// enable elevation, enable azimuth
IF MAIN.ready AND CoverControl.isopen THEN
	ElevationControl.enable := TRUE;
	AzimuthElevationControl.enable := TRUE;
	DerotatorControl.enable := TRUE;
	FilterWheelControl.Enable := TRUE;
END_IF

IF ElevationControl.Ready AND NOT ElevationControl.Calibrated THEN
	ElevationControl.HomeAxis := TRUE;
END_IF

IF AzimuthElevationControl.ready AND NOT AzimuthElevationControl.calibrated THEN
	AzimuthElevationControl.HomeAxis := TRUE;
END_IF

// enable derotator
IF ElevationControl.Ready THEN
	DerotatorControl.HomeAxis := DerotatorControl.Ready AND NOT DerotatorControl.Calibrated;
END_IF

// home filterwheel after Derotator Axis to avoid additional torque
IF DerotatorControl.Calibrated THEN
	FilterWheelControl.HomeAxis := FilterWheelControl.Ready AND NOT FilterWheelControl.Calibrated;
END_IF

// start calibration of focus after elevation has been calibrated
// this avoids imbalance by the M2 mirror on the elvation during its calibration
IF ElevationControl.Calibrated AND NOT FocusControl.Calibrated THEN
	FocusControl.enable := TRUE;
	FocusControl.HomeAxis := TRUE;
END_IF

IF CoverControl.isopen AND 
	ElevationControl.Calibrated AND
	AzimuthElevationControl.calibrated AND
	DerotatorControl.Calibrated AND
	FilterWheelControl.Calibrated AND
	FocusControl.Calibrated THEN
	power := FALSE;
	poweron := TRUE;
	isparked := FALSE;
	// rest filterwheel until reactivation on filter change
	FilterWheelControl.Enable := FALSE;
	// slew the telescope to the home position
	gohome := TRUE;
ELSE
	poweron := FALSE;
END_IF
END_METHOD

METHOD slewtelescope : USINT
VAR_INPUT
END_VAR
VAR
	SlewEvent:	FB_Eventlog;
	command_timeout: TON;
END_VAR
VAR_STAT
	Stage:		USINT := 0;
	LastStage:	USINT := 101;
END_VAR
slewtelescope := Stage;
command_timeout(IN := Stage < 100, PT := T#600S);
IF command_timeout.Q THEN
	error := TRUE;
	errorid := 16#40;
	slew := FALSE;
	Stage := 0;
END_IF
IF reset OR error THEN
	Stage := 0;
END_IF
CASE Stage OF
	0:	
		IF ready AND stopped AND NOT busy AND NOT tracking THEN
			Stage := 25;
		END_IF
	25:
		ElevationControl.position := elevation;
		ElevationControl.velocity := 10.0;
		ElevationControl.MoveAxis := TRUE;
		AzimuthElevationControl.position := azimuth;
		AzimuthElevationControl.velocity := 10.0;
		AzimuthElevationControl.MoveAxis := TRUE;
		DerotatorControl.position := elevation + derotator_offset;
		DerotatorControl.Velocity := 10.0;
		DerotatorControl.MoveAxis := TRUE;
		IF ElevationControl.ElevationAxis.Busy AND
			AzimuthElevationControl.AzimuthAxis.Busy AND
			DerotatorControl.DerotatorAxis.Busy THEN
				Stage := 50;
		END_IF
	50:
		IF ElevationControl.ElevationAxis.MoveDone THEN
			ElevationControl.MoveAxis := FALSE;
		END_IF
		
		IF AzimuthElevationControl.AzimuthAxis.MoveDone THEN
			AzimuthElevationControl.MoveAxis := FALSE;
		END_IF

		IF DerotatorControl.DerotatorAxis.MoveDone THEN
			DerotatorControl.MoveAxis := FALSE;
		END_IF
		IF NOT sliding AND stopped THEN // all axis standstill
			Stage := 100;
		END_IF
	100:
		ElevationControl.MoveAxis := FALSE;
		AzimuthElevationControl.MoveAxis := FALSE;
		DerotatorControl.MoveAxis := FALSE;
		rightascension := rightascension_calc;
		declination := declination_calc;
		slew := FALSE;
		Stage := 0;
END_CASE
SlewEvent(Trigger := Stage > LastStage, FormatString := 'Slew progress: %s', OnMessage := USINT_TO_STRING(Stage));
LastStage := Stage;
END_METHOD

METHOD stoptelescope : BOOL
VAR_INPUT
END_VAR
ElevationControl.StopAxis := TRUE;
AzimuthElevationControl.StopAxis := TRUE;
DerotatorControl.StopAxis := TRUE;
IF stopped THEN
	ElevationControl.StopAxis := FALSE;
	AzimuthElevationControl.StopAxis := FALSE;
	DerotatorControl.StopAxis := FALSE;
	stop := FALSE;
END_IF
END_METHOD

METHOD tracktelescope : BOOL
VAR_INPUT
END_VAR
// Elevation
DerotatorVelocity := F_Derotatorvelocity(elevation_calc, azimuth_calc, latitude);
ElevationVelocity := F_Elevationvelocity(azimuth_calc, latitude);
AzimuthVelocity := F_Azimuthvelocity(elevation_calc, azimuth_calc, latitude);
IF elevation_current < 5.0 OR elevation_current > 89.5 THEN 
	track := FALSE;
END_IF
IF azimuth_current > 440.0 THEN
	track := FALSE;
END_IF
IF (derotator_current < -69.0 AND DerotatorVelocity<0.0) OR (derotator_current > 379.0 AND DerotatorVelocity>0.0) THEN
	track := FALSE;
END_IF

ElevationControl.position := elevation_calc;
IF NOT ElevationControl.Tracking THEN
	ElevationControl.velocity := 10.0;
	ElevationControl.MoveAxis := TRUE;
	IF NOT ElevationControl.ElevationAxis.Busy AND ElevationControl.ElevationAxis.MoveDone THEN
		ElevationControl.MoveAxis := FALSE;
		IF ElevationControl.ElevationAxis.isTracking THEN
			ElevationControl.velocity := ElevationVelocity;
		ELSE
			ElevationControl.velocity := 3.0*ElevationVelocity;
		END_IF
		ElevationControl.velocity := ElevationVelocity;
		ElevationControl.Tracking := TRUE;
	END_IF
ELSE
	ElevationControl.velocity := ElevationVelocity;
END_IF

// Azimuth
AzimuthElevationControl.position := azimuth_calc;
IF NOT AzimuthElevationControl.Tracking THEN
	AzimuthElevationControl.velocity := 10.0;
	AzimuthElevationControl.MoveAxis := TRUE;
	IF NOT AzimuthElevationControl.AzimuthAxis.Busy AND AzimuthElevationControl.AzimuthAxis.MoveDone THEN
		AzimuthElevationControl.MoveAxis := FALSE;
		IF AzimuthElevationControl.AzimuthAxis.isTracking THEN
			AzimuthElevationControl.velocity := AzimuthVelocity;
		ELSE
			AzimuthElevationControl.velocity := 3.0*AzimuthVelocity;
		END_IF
		AzimuthElevationControl.velocity := AzimuthVelocity;
		AzimuthElevationControl.Tracking := TRUE;
	END_IF
ELSE
	AzimuthElevationControl.velocity := AzimuthVelocity;
END_IF

// Derotator
DerotatorControl.position := derotation_calc;
IF NOT DerotatorControl.Tracking THEN
	DerotatorControl.Velocity := 10.0;
	DerotatorControl.MoveAxis := TRUE;
	IF NOT DerotatorControl.DerotatorAxis.Busy AND DerotatorControl.DerotatorAxis.MoveDone THEN
		DerotatorControl.MoveAxis := FALSE;
		IF DerotatorControl.DerotatorAxis.isTracking THEN
			DerotatorControl.Velocity := DerotatorVelocity;
		ELSE
			DerotatorControl.Velocity := 3.0*DerotatorVelocity;
		END_IF
		DerotatorControl.Velocity := DerotatorVelocity;
		DerotatorControl.Tracking := TRUE;
	END_IF
ELSE
	DerotatorControl.Velocity := DerotatorVelocity;
END_IF
END_METHOD

END_PROGRAM

// ---- POUs/FunctionBlocks/FB_AstroClock.TcPOU
FUNCTION_BLOCK FB_AstroClock
VAR_INPUT
END_VAR
VAR_OUTPUT
        time_RTCEX      : DT;
        time_RTCEX2     : TIMESTRUCT;
        nMilliseconds   : DWORD;
        nMicroseconds   : DWORD;
END_VAR
VAR
	        fbGetLocalTime  : NT_GetTime;
        bBusy           : BOOL;
        bError          : BOOL;
        nErrID          : UDINT;
        presetTime      : TIMESTRUCT;

        syncTimer       : TON;
        syncTrigger     : F_TRIG;
        bSynchronize    : BOOL;

        fbRTC           : RTC;
        bValid_RTC      : BOOL;
        time_RTC        : DT;

        fbRTC_EX        : RTC_EX;
        bValid_RTCEX    : BOOL;

        fbRTC_EX2       : RTC_EX2;
        bValid_RTCEX2   : BOOL;
END_VAR

(*
TYPE TIMESTRUCT
STRUCT
   wYear            : WORD;
   wMonth           : WORD;
   wDayOfWeek       : WORD;
   wDay             : WORD;
   wHour            : WORD;
   wMinute          : WORD;
   wSecond          : WORD;
   wMilliseconds    : WORD;
END_STRUCT
END_TYPE
*)

syncTimer(IN := NOT SyncTimer.Q, PT := T#5S);
fbGetLocalTime(START := syncTimer.Q,
	TMOUT := DEFAULT_ADS_TIMEOUT,
	Busy => bBusy,
	ERR => bError,
	ERRID => nErrID,
	TIMESTR => presetTime);

syncTrigger(CLK := bBusy AND NOT bError, Q => bSynchronize);

fbRTC(EN := bSynchronize,
	PDT := SYSTEMTIME_TO_DT(presetTime),
	Q => bValid_RTC,
	CDT => time_RTC);
	
fbRTC_EX(EN := bSynchronize,
	PDT := SYSTEMTIME_TO_DT(presetTime),
	PMSEK := presetTime.wMilliseconds,
	Q => bValid_RTCEX,
	CDT => time_RTCEX,
	CMSEK => nMilliseconds);

fbRTC_EX2(EN := bSynchronize,
	PDT := presetTime,
	PMICRO := 0,
	Q => bValid_RTCEX2,
	CDT => time_RTCEX2,
	CMICRO => nMicroseconds);

END_FUNCTION_BLOCK

// ---- POUs/FunctionBlocks/FB_EQ2HOR2.TcPOU
FUNCTION_BLOCK FB_EQ2HOR2
VAR_INPUT
	// right ascension in degrees
	alpha: LREAL;
	// declination in degrees
	delta: LREAL;
	// longitude in degrees
	lon: LREAL;
	// latitude in degrees
	lat: LREAL;
	// Julian Days
	JD: LREAL;
END_VAR
VAR_OUTPUT
	// altitude in degrees
	alt: LREAL;
	// azimuth in degrees
	az: LREAL;
	// hour angle in degreesss
	ha: LREAL;
END_VAR
VAR
	lst: LREAL;
	// helper variables
	sinalt,
	// in radians
	phi_r, tau_r, alpha_r, delta_r: LREAL;
	// current epoch
	J_now: 		LREAL;
	// enable precession
	precess: 	BOOL := TRUE;
	// enable nutation
	nutate:		BOOL := TRUE;
	// enable abberation
	abberation:	BOOL := TRUE;
	// enable refraction correction
	refract:	BOOL := TRUE;
	// precession function block
	fbprecess: 	FB_PRECESS3;
	// nutation function block
	co_nutate: CO_NUTATE;
	// abberration function block
	fbaberration: CO_ABERRATION;
	//precessed coordinates
	alpha1, delta1, 
	d_alpha2, d_delta2, 
	d_alpha3, d_delta3:	LREAL;
END_VAR
VAR CONSTANT
	d2r:	LREAL := PI/180.0;
	r2d:	LREAL := 180.0/PI;
END_VAR

(* 
source: http://star-www.st-and.ac.uk/~fv/webnotes/chapter7.htm
https://squarewidget.com/astronomical-calculations-sidereal-time/

*)
lst := ct2lst(lon, jd) * 15.0; // lst in degrees

J_now := (JD - 2451545.0)/365.25 + 2000.0; // compute current equinox
IF precess THEN
	fbprecess( ra := alpha, dec := delta, 
	//EQUINOX1 := 2000.0, EQUINOX2 := J_now, 
	ra_precessed =>alpha1, dec_precessed => delta1);
ELSE
	alpha1 := alpha;
	delta1 := delta;	
END_IF

IF nutate THEN
	co_nutate(	jd := jd, 
				ra := alpha, 
				dec := delta, 
				d_ra => d_alpha2, 
				d_dec => d_delta2);
	alpha1 := alpha1 + d_alpha2;
	delta1 := delta1 + d_delta2;
ELSE
	d_alpha2 := 0.0;
	d_delta2 := 0.0;
END_IF

IF abberation THEN
	fbaberration(	jd := jd, 
					ra := alpha, 
					dec := delta, 
					d_ra => d_alpha3, 
					d_dec => d_delta3);
	alpha1 := alpha1 + d_alpha3;
	delta1 := delta1 + d_delta3;
ELSE
	d_alpha3 := 0.0;
	d_delta3 := 0.0;
END_IF

ha := MODABS(lst - alpha1, 360.0);

alpha_r := alpha1 * d2r;
delta_r := delta1 * d2r;
tau_r := lst*d2r - alpha_r;
phi_r := lat*d2r;

sinalt := SIN(phi_r)*SIN(delta_r) + COS(phi_r)*COS(delta_r)*COS(tau_r);
alt := ASIN(sinalt) * r2d;
IF refract THEN
	alt := alt + Refraction(alt, pressure := 770.0, temperature := 10.0);
END_IF
az := ATAN2(SIN(tau_r), SIN(phi_r)*COS(tau_r) - COS(phi_r)*TAN(delta_r)) * r2d + 180.0;

END_FUNCTION_BLOCK

// ---- POUs/FunctionBlocks/FB_PRECESS3.TcPOU
FUNCTION_BLOCK FB_PRECESS3
VAR_INPUT
	// right ascension in degrees
	ra: LREAL;
	// declination in degrees
	dec: LREAL;
	
END_VAR
VAR_OUTPUT
	// precessed right ascension
	ra_precessed:	LREAL;
	// precessed declination
	dec_precessed:	LREAL;
END_VAR
VAR
	ra_rad, dec_rad: LREAL;
	// starting jd (J2000)
	jd0: LREAL;
	// traget JD
	jd: LREAL;
	t, 
	eta, 
	z, 
	phi,
	A,
	B,
	C	: LREAL;
END_VAR
VAR CONSTANT
	deg_to_rad : LREAL := PI/180.0;
	sec_to_rad : LREAL := deg_to_rad/3600.0;
END_VAR

// see Jean Meeus p.135

ra_rad := ra*deg_to_rad;
dec_rad := dec*deg_to_rad;

// todo epoch to jd and jd0
JD := TelescopeControl.jd;
jd0 := 2451545.0;
t := (jd - jd0) / 36525.0;

eta :=	(2306.2181*t + 0.30188*t*t + 0.017998*t*t*t) * sec_to_rad;
z :=	(2306.2181*t + 1.09468*t*t + 0.018203*t*t*t) * sec_to_rad;
phi :=	(2004.3109*t - 0.42665*t*t - 0.041833*t*t*t) * sec_to_rad;

A :=            COS(dec_rad) * SIN(ra_rad + eta);
B := COS(phi) * COS(dec_rad) * COS(ra_rad + eta) - SIN(phi) * SIN(dec_rad);
C := SIN(phi) * COS(dec_rad) * COS(ra_rad + eta) + COS(phi) * SIN(dec_rad);

// tan(ra - z) == A/B
ra_precessed := MODABS((ATAN2(A, B) + z)/deg_to_rad, 360);
IF ABS(dec) > 89.5 THEN
	dec_precessed := ACOS(SQRT(A*A + B*B))/deg_to_rad;
ELSE
	// sin(de)c = C
	dec_precessed := ASIN(C)/deg_to_rad;	
END_IF

END_FUNCTION_BLOCK

// ---- POUs/Functions/ATAN2.TcPOU
FUNCTION ATAN2 : LREAL
VAR_INPUT
	y, x: LREAL;
END_VAR
VAR
END_VAR

(* source: https://de.wikipedia.org/wiki/Arctan2 
arctan2(y, x) := arctan(x/y)*sgn(x)^2
WARNING! The arguments are reversed compared to original wiki formula!
 *)
ATAN2 := 0.0;

IF x > 0 THEN
	ATAN2 := ATAN(y/x);
ELSIF x < 0 AND y > 0 THEN
	ATAN2 := ATAN(y/x) + PI;
ELSIF x < 0 AND y = 0 THEN
	ATAN2 := PI;
ELSIF x < 0 AND y < 0 THEN
	ATAN2 := ATAN(y/x) - PI;
ELSIF x = 0 AND y > 0 THEN
	ATAN2 := PI/2.0;
ELSIF x = 0 AND y < 0 THEN
	ATAN2 := -PI/2.0;
END_IF

END_FUNCTION

// ---- POUs/FunctionBlocks/CO_NUTATE.TcPOU
FUNCTION_BLOCK CO_NUTATE
VAR_INPUT
	// Julian date
	jd:	LREAL;
	// right ascension
	ra: LREAL;
	// declination
	dec: LREAL;
END_VAR
VAR_OUTPUT
	d_ra:	LREAL;
	d_dec:	LREAL;
	eps:	LREAL;
	d_psi:	LREAL;
END_VAR
VAR
	T, eps0, d_eps, ce, se, x,y,z, ra2, dec2: LREAL;
	x2, y2, z2:	LREAL;
	radius, xyproj: 	LREAL;
	nutate:	FB_NUTATE;
END_VAR
VAR CONSTANT
	d2r:	LREAL := PI/180.0;
	d2as: 	LREAL := PI/(180.0*3600.0);
END_VAR

 
T := (jd - 2451545.0)/36525.0; // Julian centuries FROM J2000 OF jd.

// must calculate obliquity of ecliptic
nutate(jd := jd, nut_long => d_psi, nut_obliq => d_eps );

eps0 := 23.4392911*3600.0 - 46.8150*T - 0.00059*T*T + 0.001813*T*T*T;
eps := (eps0 + d_eps)/3600.0*d2r; // true obliquity of the ecliptic in radians
 
//useful numbers
ce := COS(eps);
se := SIN(eps);

// convert ra-dec to equatorial rectangular coordinates
x := COS(ra*d2r) * COS(dec*d2r);
y := SIN(ra*d2r) * COS(dec*d2r);
z := SIN(dec*d2r);

// apply corrections to each rectangular coordinate
x2 := x - (y*ce + z*se)*d_psi * d2as;
y2 := y + (x*ce*d_psi - z*d_eps) * d2as;
z2 := z + (x*se*d_psi + y*d_eps) * d2as;

// convert back to equatorial spherical coordinates
radius := SQRT(x2*x2 + y2*y2 + z2*z2);
xyproj := SQRT(x2*x2 + y2*y2);

ra2 := x2 * 0.0;
dec2:= x2 * 0.0;
// Calculate Ra and Dec in RADIANS (later convert to DEGREES)

IF xyproj = 0.0 AND z <> 0.0 THEN
	// places where xyproj:=0 (point at NCP or SCP)
	dec2 := ASIN(z2/radius);
	ra2 := 0.0;
END_IF
IF xyproj <> 0.0 THEN
	ra2 := ATAN2(y2, x2);
	dec2 := ASIN(z2 / radius);
END_IF

// convert to DEGREES
ra2 := ra2 /d2r;
dec2 := dec2 /d2r;

// w := where(ra2 LT 0., Nw)
// IF Nw GT 0 THEN ra2[w] := ra2[w] + 360.
ra2 := MODABS(ra2, 360.0);

// Return changes in ra and dec in degrees
 d_ra := ra2 - ra;
 d_dec := dec2 - dec;

END_FUNCTION_BLOCK

// ---- POUs/FunctionBlocks/FB_NUTATE.TcPOU
FUNCTION_BLOCK FB_NUTATE
VAR_INPUT
	jd:	LREAL;
END_VAR
VAR_OUTPUT
	nut_long, nut_obliq: LREAL := 0.0;
END_VAR
VAR
	t: LREAL;
	d, M, Mprime, F, omega: LREAL;
	arg, sarg, carg:  ARRAY[0..62] OF LREAL;
	I: INT;
END_VAR
VAR CONSTANT
	dtor:	LREAL := PI/180.0;
	coeff1:	ARRAY[0..3] OF LREAL := [297.85036, 445267.111480, -0.0019142,  1.0/189474];
	coeff2:	ARRAY[0..3] OF LREAL := [357.52772,  35999.050340, -0.0001603, -1.0/3E5]; 
	coeff3:	ARRAY[0..3] OF LREAL := [134.96298, 477198.867398,  0.0086972,  1.0/5.625E4]; 
	coeff4:	ARRAY[0..3] OF LREAL :=  [93.27191, 483202.017538, -0.0036825, -1.0/3.27270E5]; 
  	coeff5: ARRAY[0..3] OF LREAL := [125.04452,  -1934.136261,  0.0020708,  1.0/4.5E5];
	d_lng: ARRAY[0..62] OF LREAL := [0,-2,0,0,0,0,-2,0,0,-2,-2,-2,0,2,0,2,0,0,-2,0,2,0,0,-2,0,-2,0,0,2,-2,0,-2,0,0,2,2,0,-2,0,2,2,-2,-2,2,2,0,-2,-2,0,-2,-2,0,-1,-2,1,0,0,-1,0,0,2,0,2]; 
	m_lng: ARRAY[0..62] OF LREAL := [0,0,0,0,1,0,1,0,0,-1,17(0),2,0,2,1,0,-1,0,0,0,1,1,-1,0,0,0,0,0,0,-1,-1,0,0,0,1,0,0,1,0,0,0,-1,1,-1,-1,0,-1];
	mp_lng: ARRAY[0..62] OF LREAL := [0,0,0,0,0,1,0,0,1,0,1,0,-1,0,1,-1,-1,1,2,-2,0,2,2,1,0,0,-1,0,-1,0,0,1,0,2,-1,1,0,1,0,0,1,2,1,-2,0,1,0,0,2,2,0,1,1,0,0,1,-2,1,1,1,-1,3,0];
	f_lng: ARRAY[0..62] OF LREAL := [0,2,2,0,0,0,2,2,2,2,0,2,2,0,0,2,0,2,0,2,2,2,0,2,2,2,2,0,0,2,0,0,0,-2,2,2,2,0,2,2,0,2,2,0,0,0,2,0,2,0,2,-2,0,0,0,2,2,0,0,2,2,2,2];
	om_lng: ARRAY[0..62] OF LREAL := [1,2,2,2,0,0,2,1,2,2,0,1,2,0,1,2,1,1,0,1,2,2,0,2,0,0,1,0,1,2,1,1,1,0,1,2,2,0,2,1,0,2,1,1,1,0,1,1,1,1,1,0,0,0,0,0,2,0,0,2,2,2,2];
	sin_lng: ARRAY[0..62] OF LREAL := [-171996, -13187, -2274, 2062, 1426, 712, -517, -386, -301, 217, -158, 129, 123, 63, 63, -59, -58, -51, 48, 46, -38, -31, 29, 29, 26, -22, 21, 17, 16, -16, -15, -13, -12, 11, -10, -8, 7, -7, -7, -7, 6,6,6,-6,-6,5,-5,-5,-5,4,4,4,-4,-4,-4,3,-3,-3,-3,-3,-3,-3,-3 ];
	sdelt: ARRAY[0..62] OF LREAL := [-174.2, -1.6, -0.2, 0.2, -3.4, 0.1, 1.2, -0.4, 0, -0.5, 0, 0.1, 0,0,0.1, 0,-0.1,10(0), -0.1, 0, 0.1, 33(0)];
	cos_lng: ARRAY[0..62] OF LREAL := [ 92025, 5736, 977, -895, 54, -7, 224, 200, 129, -95,0,-70,-53,0, -33, 26, 32, 27, 0, -24, 16,13,0,-12,0,0,-10,0,-8,7,9,7,6,0,5,3,-3,0,3,3, 0,-3,-3,3,3,0,3,3,3, 14(0)] ;
	cdelt: ARRAY[0..62] OF LREAL := [8.9, -3.1, -0.5, 0.5, -0.1, 0.0, -0.6, 0.0, -0.1, 0.3, 53(0)];
END_VAR

//  form time in Julian centuries from 1900.0

t := (jd - 2451545.0)/36525.0;

// Mean elongation of the Moon

d := poly(T, coeff1)*dtor;
d := MODABS(d, 2.0*PI);

// Sun's mean anomaly

M := poly(T,coeff2)*dtor;
M := MODABS(M, 2.0*PI);

// Moon's mean anomaly

Mprime := poly(T,coeff3)*dtor;
Mprime := MODABS(Mprime, 2.0*PI);

// Moon's argument of latitude

F := poly(T, coeff4 )*dtor;
F := MODABS(F, 2.0*PI);

// Longitude OF the ascending node OF the Moon's mean orbit on the ecliptic,
//  measured from the mean equinox of the date

omega := poly(T, coeff5)*dtor;
omega := MODABS(omega, 2.0*PI);


// Sum the periodic terms 
FOR i:=0 TO 62 DO
	arg[i] := d_lng[i]*d + m_lng[i]*m +mp_lng[i]*mprime + f_lng[i]*f +om_lng[i]*omega;
	sarg[i] := SIN(arg[i]);
	carg[i] := COS(arg[i]);
END_FOR

nut_long  := 0.0;
nut_obliq := 0.0;

FOR i:=0 TO 62 DO
	nut_long  := nut_long  + 0.0001*( (sdelt[i]*t + sin_lng[i])*sarg[i]);
	nut_obliq := nut_obliq + 0.0001*( (cdelt[i]*t + cos_lng[i])*carg[i]);
END_FOR

END_FUNCTION_BLOCK

// ---- POUs/Functions/POLY.TcPOU
FUNCTION POLY : LREAL
VAR_INPUT
	X:	LREAL;
	COEFFS: ARRAY [0..3] OF LREAL;
END_VAR
VAR
END_VAR

POLY := COEFFS[0]*EXPT(X, 0) + COEFFS[1]*EXPT(X, 1) + COEFFS[2]*EXPT(X, 2) + COEFFS[3]*EXPT(X, 3);

END_FUNCTION

// ---- POUs/FunctionBlocks/CO_ABERRATION.TcPOU
FUNCTION_BLOCK CO_ABERRATION
VAR_INPUT
	jd, 				// Julian Date
	ra, dec: LREAL; 	//ra and dec in degrees
	eps : LREAL := 0.0;
END_VAR
VAR_OUTPUT
	d_ra, d_dec: LREAL;
END_VAR
VAR
	sunpos: FB_SUNPOS;
	nutate: FB_NUTATE;
	sunra, sundec, sunlon,
	d_psi, d_epsilon, eps0,
	t, e, peri, cd, sd, ce, te, cp, sp, cs, ss, ca, sa, term1, term2, term3, term4: LREAL;
END_VAR
VAR CONSTANT
	d2r : LREAL := PI/180.0;
	k: LREAL := 20.49552; //constant of aberration, in arcseconds
	
END_VAR

(*
;+
;  NAME:
;     CO_ABERRATION
; PURPOSE:
;     Calculate changes to Ra and Dec due to the effect of annual aberration 
; EXPLANATION:
;      as described in Meeus, Chap 23.
; CALLING SEQUENCE:
;      co_aberration, jd, ra, dec, d_ra, d_dec, [EPS = ]
; INPUTS
;       jd      : Julian Date [scalar or vector]
;       ra, dec : Arrays (or scalars) of the ra  and dec's in degrees
;   Note: if jd is a vector, then ra and dec must either be scalars, or 
;                vectors of the same length.
;
; OUTPUTS
;       d_ra, d_dec: the corrections to ra and dec due to aberration in 
;                    arcseconds.  (These values can be added to the true RA 
;                    and dec to get the apparent position).   Note that d_ra
;                     is *not* multiplied by cos(dec), so that 
;                     apparent_ra = ra + d_ra/3600. 
; OPTIONAL INPUT KEYWORD:
;       eps : set this to the true obliquity of the ecliptic (in radians), or
;         it will be set for you if you don't know it (in that case, set it to
;                 an empty variable).
; EXAMPLE:
;   Compute the change in RA and Dec of Theta Persei (RA = 2h46m,11.331s, Dec =
;   49d20',54.54") due to aberration on 2028 Nov 13.19 TD
;
;      IDL> jdcnv,2028,11,13,.19*24,jd      ;Get Julian date
;      IDL> co_aberration,jd,ten(2,46,11.331)*15,ten(49,20,54.54),d_ra,d_dec
;
;      ==> d_ra = 30.045" (=2.003s)    d_dec = 6.697"
; NOTES:
;  These formula are from Meeus, Chapters 23.  Accuracy is much better than 1 
;   arcsecond.
;
;   The maximum deviation due to annual aberration is 20.49" and occurs when the
;   Earth velocity is perpendicular to the direction of the star.
;
; REVISION HISTORY:
;   Written, June 2002,      Chris O'Dell, U. of Wisconsin
;   Fix error with vector input   W. Landsman   June 2009
;   June 2009 update fixed case where JD was scalar but RA,Dec were vectors, but 
;     broke the case when both JD and RA,Dec were vectors Aug 2012 W. Landsman
;   Further fix when JD is 1 element vector  W. Landsman
;-
*)

T := (jd -2451545.0)/36525.0; // julian centuries from J2000 of jd.

IF EPS = 0.0 THEN
	// must calculate obliquity of ecliptic
	nutate(jd := jd, nut_long => d_psi, nut_obliq => d_epsilon); //d_psi and d_epsilon in degrees
	eps0 := ten(23,26,21.448)*3600.0 - 46.8150*T - 0.00059*EXPT(T, 2) +  0.001813*EXPT(T, 3);
	// TRUE obliquity OF the ecliptic in radians
	eps := (eps0 + d_epsilon)/3600.0*d2r; 	
END_IF

sunpos( JD := jd, RA => sunra, Dec => sundec, longmed => sunlon);

// Earth's orbital eccentricity
e := 0.016708634 - 0.000042037*T - 0.0000001267*EXPT(T, 2);
// longitude of perihelion, in degrees 
peri := 102.93735 + 1.71946*T + 0.00046*EXPT(T, 2);

//Useful Trig Functions
cd := COS(dec*d2r);		sd := SIN(dec*d2r);
ce := COS(eps); 		te := TAN(eps);
cp := COS(peri*d2r);	sp := SIN(peri*d2r);
cs := COS(sunlon*d2r);	ss := SIN(sunlon*d2r);
ca := COS(ra*d2r);		sa := SIN(ra*d2r);

term1 := (ca*cs*ce + sa*ss)/cd;
term2 := (ca*cp*ce + sa*sp)/cd;
term3 := (cs*ce*(te*cd - sa*sd) + ca*sd*ss);
term4 := (cp*ce*(te*cd - sa*sd) + ca*sd*sp);

d_ra := (-k * term1 + e*k * term2)/3600.0;
d_dec := (-k * term3 + e*k * term4)/3600.0;

END_FUNCTION_BLOCK

// ---- POUs/FunctionBlocks/FB_SUNPOS.TcPOU
FUNCTION_BLOCK FB_SUNPOS
VAR_INPUT
	// Julian Date
	JD:		LREAL;
	// output in Radians instead of Degrees
	RADIAN:	BOOL:= FALSE;
END_VAR
VAR_OUTPUT
	// right ascension
	RA,
	// declination of the sun
	Dec,
	// longitude
	longmed,
	// True Obliquity
	oblt:	LREAL;
END_VAR
VAR
	t, //  Julian centuries FROM 1900.0
	l, //  sun's mean longitude
	me, // Earth's mean anomaly
	ellcor, // ellipticity of the orbit
	mv, // mean anomaly of Venus
	vencorr,
	mm, 
	marscorr,
mj, jupcorr,
d, longterm, mooncorr,  omega:	LREAL;
END_VAR
VAR CONSTANT
	dtor: LREAL := PI/180.0; // Pi/180
END_VAR

(* source: https://idlastro.gsfc.nasa.gov/ftp/pro/astro/sunpos.pro *)

//  form TIME in Julian centuries FROM 1900.0
t := (jd - 2415020.0)/36525.0;

//  form sun's mean longitude
l := (279.696678+LMOD(36000.768925*t, 360.0))*3600.0;

//  allow for ellipticity of the orbit (equation of centre) using the Earth's mean anomaly ME
me := 358.475844 + LMOD(35999.049750*t, 360.0);
ellcor  := (6910.1 - 17.2*t)*SIN(me*dtor) + 72.3*SIN(2.0*me*dtor);
l := l + ellcor;
 
// allow FOR the Venus perturbations using the mean anomaly OF Venus MV
mv := 212.603219 + LMOD(58517.803875*t, 360.0);
vencorr := 4.8 * COS((299.1017 + mv - me)*dtor) + 
          5.5 * COS((148.3133 +  2.0 * mv  -  2.0 * me )*dtor) + 
          2.5 * COS((315.9433 +  2.0 * mv  -  3.0 * me )*dtor) + 
          1.6 * COS((345.2533 +  3.0 * mv  -  4.0 * me )*dtor) + 
          1.0 * COS((318.15   +  3.0 * mv  -  5.0 * me )*dtor);
l := l + vencorr;

//  Allow FOR the Mars perturbations using the mean anomaly OF Mars MM
mm := 319.529425  +  LMOD( 19139.858500 * t,  360.0 );
marscorr := 2.0 * COS((343.8883 -  2.0 * mm  +  2.0 * me)*dtor ) + 
            1.8 * COS((200.4017 -  2.0 * mm  + me) * dtor);
l := l + marscorr;

// Allow FOR the Jupiter perturbations using the mean anomaly OF Jupiter MJ
mj := 225.328328  +  LMOD( 3034.6920239 * t,  360.0 );
jupcorr := 7.2 * COS(( 179.5317 - mj + me )*dtor) + 
          2.6 * COS((263.2167  -  MJ ) *dtor) + 
          2.7 * COS(( 87.1450  -  2.0 * mj  +  2.0 * me ) *dtor) + 
          1.6 * COS((109.4933  -  2.0 * mj  +  me ) *dtor);
l := l + jupcorr;

// Allow FOR the Moons perturbations using the mean elongation OF the Moon from the Sun D
d := 350.7376814  + LMOD( 445267.11422 * t,  360.0 );
mooncorr  := 6.5 * SIN(d*dtor);
l := l + mooncorr;

// Allow for long period terms
longterm := 6.4 * SIN(( 231.19  +  20.20 * t )*dtor);
l :=  l + longterm;
l :=  LMOD( l + 2592000.0,  1296000.0); 
longmed := l/3600.0;

// Allow for Aberration
l :=  l - 20.5;

// Allow for Nutation using the longitude of the Moons mean node OMEGA
omega := 259.183275 - LMOD( 1934.142008 * t, 360.0);
l :=  l - 17.2 * SIN(omega*dtor);

// Form the True Obliquity
oblt := 23.452294 - 0.0130125*t + (9.2*COS(omega*dtor))/3600.0;

// Form Right Ascension AND Declination
l := l/3600.0;
ra := ATAN2( SIN(l*dtor) * COS(oblt*dtor), COS(l*dtor));
//ra := MODABS(ra, 360.0);
dec := ASIN(SIN(l*dtor) * SIN(oblt*dtor));
 
IF RADIAN THEN
	oblt := oblt*dtor; 
	longmed := longmed*dtor;
ELSE
	ra := ra/dtor;
    dec := dec/dtor;
END_IF

END_FUNCTION_BLOCK

// ---- POUs/Functions/CT2LST.TcPOU
FUNCTION CT2LST : LREAL
VAR_INPUT
	lng: LREAL; // The longitude in degrees (east of Greenwich) of the place for which the local sidereal time is desired, scalar.   The Greenwich mean sidereal time (GMST) can be found by setting Lng = 0.
	jd:	LREAL; // this is the Julian date of time in question
END_VAR
VAR
	t0,t,theta: LREAL;
END_VAR
VAR CONSTANT
	jd2000: LREAL := 2451545.0;
END_VAR

(* source https://idlastro.gsfc.nasa.gov/ftp/pro/astro/ct2lst.pro 

;+
; NAME:
;     CT2LST
; PURPOSE:
;     To convert from Local Civil Time to Local Mean Sidereal Time.
;
; CALLING SEQUENCE:
;     CT2LST, Lst, Lng, Tz, Time, [Day, Mon, Year] 
;                       or
;     CT2LST, Lst, Lng, dummy, JD
;
; INPUTS:
;     Lng  - The longitude in degrees (east of Greenwich) of the place for 
;            which the local sidereal time is desired, scalar.   The Greenwich 
;            mean sidereal time (GMST) can be found by setting Lng = 0.
;     Tz  - The time zone of the site in hours, positive East  of the Greenwich
;           meridian (ahead of GMT).  Use this parameter to easily account 
;           for Daylight Savings time (e.g. -4=EDT, -5 = EST/CDT), scalar
;           This parameter is not needed (and ignored) if Julian date is 
;           supplied.    ***Note that the sign of TZ was changed in July 2008
;           to match the standard definition.*** 
;     Time or JD  - If more than four parameters are specified, then this is 
;               the time of day of the specified date in decimal hours.  If 
;               exactly four parameters are specified, then this is the 
;               Julian date of time in question, scalar or vector
;
; OPTIONAL INPUTS:
;      Day -  The day of the month (1-31),integer scalar or vector
;      Mon -  The month, in numerical format (1-12), integer scalar or vector
;      Year - The 4 digit year (e.g. 2008), integer scalar or vector
;
; OUTPUTS:
;       Lst   The Local Sidereal Time for the date/time specified in hours.
;
; RESTRICTIONS:
;       If specified, the date should be in numerical form.  The year should
;       appear as yyyy.
;
; PROCEDURE:
;       The Julian date of the day and time is question is used to determine
;       the number of days to have passed since 0 Jan 2000.  This is used
;       in conjunction with the GST of that date to extrapolate to the current
;       GST; this is then used to get the LST.    See Astronomical Algorithms
;       by Jean Meeus, p. 84 (Eq. 11-4) for the constants used.
;
; EXAMPLE:
;       Find the Greenwich mean sidereal time (GMST) on 2008 Jul 30 at 15:53 pm
;       in Baltimore, Maryland (longitude=-76.72 degrees).   The timezone is 
;       EDT or tz=-4
;
;       IDL> CT2LST, lst, -76.72, -4,ten(15,53), 30, 07, 2008
;
;               ==> lst =  11.356505  hours  (= 11h 21m 23.418s)
;
;       The Web site  http://tycho.usno.navy.mil/sidereal.html contains more
;       info on sidereal time, as well as an interactive calculator.
; PROCEDURES USED:
;       jdcnv - Convert from year, month, day, hour to julian date
;
; MODIFICATION HISTORY:
;     Adapted from the FORTRAN program GETSD by Michael R. Greason, STX, 
;               27 October 1988.
;     Use IAU 1984 constants Wayne Landsman, HSTX, April 1995, results 
;               differ by about 0.1 seconds  
;     Longitudes measured *east* of Greenwich   W. Landsman    December 1998
;     Time zone now measure positive East of Greenwich W. Landsman July 2008
;     Remove debugging print statement  W. Landsman April 2009
;-

*)

t0 := jd - jd2000;
t := t0/36525.0;
// Compute GST in seconds.
theta := 280.46061837 + (360.98564736629 * t0) + EXPT(t, 2)*(0.000387933 - (t/ 3871.0E4));
//theta := 100.46061837 + 36000.770053608*t0 + 0.000387933*EXPT(t0,2) - EXPT(t0,3)/3871000.0;
// Compute LST in hours.
CT2LST := ( theta + lng)/15.0;
CT2LST := MODABS(CT2LST, 24.0);

END_FUNCTION

// ---- POUs/Functions/Refraction.TcPOU
FUNCTION Refraction : LREAL
VAR_INPUT
	// elevation in degrees
	elevation: LREAL;
	// pressure in mBar
	pressure: LREAL := 770.0;
	// temperature in Celsius
	temperature : LREAL := 10.0;
END_VAR
VAR
END_VAR
VAR CONSTANT
	d2r:	LREAL := PI/180.0;
END_VAR

// sanity checks
elevation := LIMIT(0.0, elevation, 90.0);
pressure := LIMIT(600.0, pressure, 1200.0);
temperature := LIMIT(-30.0, temperature, 40.0);
// refraction in arcmin
Refraction := 1.02 / TAN((elevation + 10.3/(elevation + 5.11)) * d2r);
Refraction := Refraction * pressure * 283.0 / (1010.0 * (273.0 + temperature));
//refraction in degrees
Refraction := Refraction / 60.0;

END_FUNCTION

// ---- POUs/FunctionBlocks/FB_HOR2EQ.TcPOU
FUNCTION_BLOCK FB_HOR2EQ
VAR_INPUT
	//altitude (in degrees) [scalar OR vector]
	alt: LREAL;  
	//azimuth angle (in degrees, measured EAST from NORTH, but see keyword WS below.) [scalar or vector]
	az: LREAL;
	// Julian Date [scalar or vector], double precision
	JD: 		LREAL;
	lat:		LREAL;
	lon:		LREAL;
	WS:			BOOL;
	precess:	BOOL := FALSE;
	NUTATE:		BOOL := FALSE;
	aberration:	BOOL := FALSE;
	refract:	BOOL := FALSE;
	altitude:	LREAL := 0.0;
END_VAR
VAR_OUTPUT
	// Right Ascension of object  (J2000) in degrees (FK5)
	ra: 	LREAL;
	// Declination of object (J2000) in degrees (FK5)
	dec:	LREAL;
	// hour angle (in degrees) (optional)
	ha:		LREAL;
END_VAR
VAR
	
	alt_,
	az_,
	lmst,
	J_now: LREAL;
	co_nutate: 		FB_CO_NUTATE;
	co_aberration: 	CO_ABERRATION;
	co_refract:		CO_REFRACT;
	fbprecess:		FB_PRECESS;
	altaz2hadec:	FB_ALTAZ2HADEC;
	last: LREAL;
	dra1: LREAL;
	ddec1: LREAL;
	eps: LREAL;
	d_psi: LREAL;
	dra2: LREAL;
	ddec2: LREAL;
END_VAR
VAR CONSTANT
	//d2r:	LREAL := PI/180.0;
	//r2d:	LREAL := 180.0/PI;
	//h2r:	LREAL := PI/12.0;
	h2d:	LREAL := 15.0;
END_VAR



alt_ := alt;   //do this so we don't change ra, dec arrays.
az_ := az;


//*******************************************************************************************
// Make Correction for ATMOSPHERIC REFRACTION
// (use this for visible and radio wavelengths; author is unsure about other wavelengths)
IF refract THEN 
	co_refract(	old_alt := alt, 
				altitude := altitude, 
				to_observed := TRUE, 
				new_alt => alt);
END_IF

IF WS THEN 
	az_ := az_ - 180.0;
END_IF

co_nutate(	jd := jd, 
			ra := 45.0, 
			dec := 45.0, 
			d_ra => dra1, 
			d_dec => ddec1, 
			eps => eps, 
			d_psi => d_psi);
//******************************************************************************
//Calculate LOCAL APPARENT SIDEREAL TIME
// first get local mean sidereal time (lmst)
// get LST (in hours) - note:this is indep of tzone since giving jd
lmst := ct2lst( lon, jd);
// convert LMST TO degrees (btw, THIS is the RA OF the zenith)
lmst := lmst*h2d;
// calculate local APPARENT sidereal time (last)
// ADD correction in degrees
last := lmst + d_psi *COS(eps)/3600.0 ; 

//****************************************************************************
// Now do the spherical trig to get APPARENT Hour Angle [degrees], and
// declination [degrees].
altaz2hadec( alt := alt_, az := az_, lat := lat, ha => ha, dec => dec);

// Find Right Ascension (in degrees, from 0 to 360.)
 ra := MODABS(last - ha + 360.0, 360.0);



//*****************************************************************************
// calculate NUTATION and ABERRATION Corrections to Ra-Dec
IF NUTATE THEN
	co_nutate(	jd := jd, 
			ra := ra, 
			dec := dec, 
			d_ra => dra1, 
			d_dec => ddec1, 
			eps => eps, 
			d_psi => d_psi);
ELSE
	dra1 := 0.0;
	ddec1 := 0.0;	
END_IF
IF aberration THEN
	co_aberration(	jd := jd, 
				ra := ra, 
				dec := dec, 
				d_ra => dra2, 
				d_dec => ddec2, 
				eps := eps);
ELSE
	dra2 := 0.0;
	ddec2 := 0.0;	
END_IF
//******************************************************************************
// Make Nutation and Aberration Corrections (if wanted)

ra := ra - (dra1 + dra2)/3600.0;
dec := dec - (ddec1 + ddec2)/3600.0;
 //compute current equinox
J_now := (JD - 2451545.0)/365.25 + 2000.0 ;

//*****************************************************************************
// PRECESS coordinates to current date
// (uses astro lib procedure PRECESS.pro)

IF precess THEN 
	fbprecess( ra := ra, dec := dec, 
	EQUINOX1 := J_now, EQUINOX2 := 2000.0, // bugfix from randnotizlukas
	ra_precessed =>ra, dec_precessed => dec);                   
END_IF

END_FUNCTION_BLOCK

// ---- POUs/Functions/DateTime2JD.TcPOU
FUNCTION DateTime2JD : LREAL
VAR_INPUT
	epoch: TIMESTRUCT;
END_VAR
VAR
	a,y,m,d,jdn: LREAL;
END_VAR

(*    import datetime
    from math import floor
    if not type(epoch) is datetime.datetime:
        raise TypeError('datetime must be of type datetime')
    
    a = floor((14 - epoch.month)/12)
    y = epoch.year + 4800 - a
    m = epoch.month + 12*a - 3
    
    d = epoch.day
    d += epoch.hour/24. + epoch.minute/1440. + epoch.second/86400. # microsecond might be added here?
    
    if [epoch.year,epoch.month,d] >= [1582,10,15]:
        jdn = epoch.day + floor((153*m + 2)/5) + 365*y + floor(y/4) - floor(y/100) + floor(y/400) - 32045
    elif [epoch.year,epoch.month,d] <= [1582,10,4]:
        jdn = epoch.day + floor((153*m + 2)/5) + 365*y + floor(y/4) - 32083
    return jdn + (epoch.hour-12)/24. + epoch.minute/1440. + epoch.second/86400.
*)
a := FLOOR((14.0 - epoch.wMonth)/12.0);
y := epoch.wYear + 4800.0 - a;
m := epoch.wMonth + 12.0*a - 3.0;

d := epoch.wDay + (epoch.wHour/24.0) + (epoch.wMinute/1440.0) + (epoch.wSecond/86400.0);

//IF (epoch.wYear > 1582) (* AND (epoch.wMonth > 10.0) AND (d > 15.0)*) THEN
	jdn := epoch.wDay + FLOOR((153*m + 2)/5) + 365.0*y + FLOOR(y/4) - FLOOR(y/100) + FLOOR(y/400) - 32045.0;
//ELSIF (epoch.wYear < 1582) AND (epoch.wMonth < 10) AND (d > 4.0) THEN
//	jdn := epoch.wDay + FLOOR((153*m + 2)/5) + 365.0*y + FLOOR(y/4) - 32083.0;
//END_IF

DateTime2JD := jdn
			+ (epoch.wHour-12.0)/24.0
			+ (epoch.wMinute/1440.0) 
			+ (epoch.wSecond/86400.0)
			+ (DWORD_TO_LREAL(epoch.wMilliseconds)/86400000.0);

END_FUNCTION

// ---- POUs/ElevationControl.TcPOU
PROGRAM ElevationControl
VAR_INPUT
	// enable the axis
	enable: 	BOOL;
	// reset an error
	reset:		BOOL;
	// increase the eleveation
	up:			BOOL;
	// decrease the elevation
	down:		BOOL;
	// set position of the axis in degrees
	position:	LREAL;
	// set the Velocity of the axis
	velocity:	LREAL;
	// move axis command
	MoveAxis:	BOOL;
	// calibrate the axis
	HomeAxis:	BOOL;
	// enable tracking
	Tracking:	BOOL;
	// stop the Axis
	StopAxis:	BOOL;
	// reset diagnostic errors
	bSoEReset:	 	BOOL;
END_VAR
VAR_OUTPUT
	// axis is ready to operate
	Ready:			BOOL;
	// drive error condition
	error: 			BOOL;
	// warning condition
	warning:		BOOL;
	// actual position of the elevation axis
	actual_position: 	LREAL;
	// error ID of the elevation axis
	ErrorID: 		UDINT;
	// axis is calibrated
	Calibrated:		BOOL;
	// time to reach target position
	slewtime:		LREAL;
END_VAR
VAR
	ElevationAxis:			FB_Axis2;
	ElevationCalibration: 	MC_SetPosition;
	fbSoEReset: 			FB_SoEReset;
	// delay until commutator angle is measured
	readydelay:				TON;
	// disable trigger for hydraulics
	enable_trigger:			F_TRIG;
	// store last position
	getlastposition:		BOOL := TRUE;
	ElevationAxisEvent: 	FB_Eventlog;
	ElevationDiagnosticEvent: 	FB_Eventlog;
	ElevationBrakeEvent: 	FB_Eventlog;
	HighElevationEvent: 	FB_Eventlog;
	LowElevationEvent:		FB_Eventlog;
	TorqueWarning:			FB_EventLog;
	CalibrationEvent:		FB_Eventlog;
	// elevation torque in percent
	elevation_torque: 		REAL;
	// timer to trigger a warning if torque is high
	torque_timer:			TON;
	ReadParameter:			MC_ReadParameter;
	DiagnosticError:		BOOL;
END_VAR
VAR CONSTANT
	// current position of the calibration cam. Apply an offset here if necessary
	calibration_position:	LREAL := 44.144 - 0.00516; //44.144; //44.139; //44.061; //43.806122; //42.1281; //43.000 | calibration_position = calibration_position - EOFF
END_VAR
VAR PERSISTENT
	last_position:	LREAL := -1.0;
END_VAR

// limit the position input to a sane value
position := LIMIT(0.0, position, 90.0);

IF Calibrated AND (actual_position > 89.0 OR actual_position < 1.0) THEN
	Tracking := FALSE;
END_IF

//if we enable the axis, we have to open the brake first
IF Enable THEN
	IF NOT Calibrated THEN
		CoverControl.open := TRUE;
		IF CoverControl.isopen THEN
			HydraulicsControl.open_brake();
		END_IF
	ELSE
		HydraulicsControl.open_brake();
	END_IF
	
END_IF

enable_trigger(CLK := enable);
// close the brake on the falling edge of the enable signal
IF enable_trigger.Q THEN
	HydraulicsControl.close_brake();
END_IF

IF ElevationAxis.Calibrated OR Error THEN
	HomeAxis := FALSE;
END_IF

Calibrated := ElevationAxis.Calibrated;

IF HomeAxis THEN
	position := calibration_position;
	MoveAxis := FALSE;
	Tracking := FALSE;
END_IF

IF MoveAxis OR StopAxis THEN
	Tracking := FALSE;
END_IF

// if NOT Enabled and ActVelo>1 then issue a warning
warning := NOT enable AND GVL_Telescope.ElevationAxisRef.NcToPlc.ActVelo>2.0;

// deactivate limit switches on homing
MC_SetAcceptBlockedDriveSignal(
	Axis := GVL_Telescope.ElevationAxisRef, 
	Enable := HomeAxis);
	
ElevationAxis(
	Enable := 			enable AND HydraulicsControl.brake_open,
	Reset := 			reset,
	MoveAxis :=			MoveAxis,
	HomeAxis :=			HomeAxis,
	StopAxis :=			StopAxis,
	Tracking :=			Tracking,
	Position := 		position, 
	Velocity :=			Velocity,
	Enable_Positive :=  GVL_Telescope.Elevation_inputs.0 OR HomeAxis,
	Enable_Negative := 	GVL_Telescope.Elevation_inputs.1,
	Jog_Forward :=		up,
	Jog_Backwards := 	down,
	bCalibrationCam :=	NOT GVL_Telescope.Elevation_inputs.0,
	ActualPosition => 	actual_position,
	Error => 			error,
	ErrorID => 			ErrorID,
	AxisRef :=			GVL_Telescope.ElevationAxisRef);

IF ElevationAxis.MoveDone THEN
	MoveAxis := FALSE;
END_IF

IF ElevationAxis.HomeDone THEN
	HomeAxis := FALSE;
END_IF
	
IF ElevationAxis.ResetDone THEN
	reset := FALSE;
END_IF

IF ElevationAxis.StopDone THEN
	StopAxis := FALSE;
END_IF

DiagnosticError := FALSE;
IF GVL_Telescope.Elevation_diagnostic < 16#D012 AND GVL_Telescope.Elevation_diagnostic > 16#D014 THEN
	DiagnosticError :=TRUE;
	ErrorID := GVL_Telescope.Elevation_diagnostic;
END_IF

ElevationCalibration(Axis := GVL_Telescope.ElevationAxisRef,
	Execute := getlastposition AND last_position>=0.0 AND NOT Calibrated,
	Position := last_position);

IF ElevationCalibration.Done THEN
	getlastposition := FALSE;
END_IF

IF Calibrated THEN
	last_position := actual_position;
END_IF

IF bSoEReset THEN
	last_position := -1.0;
	fbSoEReset(
		Axis := GVL_Telescope.ElevationAxisRef,
		Execute := TRUE,
		Timeout := DEFAULT_ADS_TIMEOUT);
 	IF NOT fbSoEReset.Busy THEN
		fbSoEReset(Axis := GVL_Telescope.ElevationAxisRef, Execute := FALSE);
		bSoEReset := FALSE;
		Reset := TRUE;
	END_IF
END_IF 

readydelay(IN :=  HydraulicsControl.brake_open, PT := T#6000MS, Q=> ready);

ReadParameter(	Axis := GVL_Telescope.ElevationAxisRef, 
				Enable := ElevationAxis.InMotion, 
				ParameterNumber := MC_AxisParameter.AxisRemainingTimeToGo, 
				ReadMode := E_ReadMode.READMODE_CYCLIC);
				
IF ReadParameter.Valid THEN
	slewtime := ReadParameter.Value;
END_IF

elevation_torque := GVL_Telescope.Elevation_torque / 10.0;
torque_timer(IN := ABS(elevation_torque) > 50.0, PT := T#1000MS);
		
ElevationAxisEvent(	Trigger := Error, 
				Level := ADSLOG_MSGTYPE_ERROR,
				FormatString := 'Elevation Axis Error: %s',
				OnMessage := NCError_TO_STRING(ErrorID));

ElevationDiagnosticEvent(	
	Trigger := 		DiagnosticError, 
	Level := 		ADSLOG_MSGTYPE_ERROR,
	FormatString :=	'Elevation Axis Diagnostic Error: %s',
	OnMessage := 	NCError_TO_STRING(GVL_Telescope.Elevation_diagnostic));

				
HighElevationEvent(	Trigger := Calibrated AND actual_position > 85.0, 
				Level := ADSLOG_MSGTYPE_WARN,
				FormatString := 'High Elevation: %s',
				OnMessage := LREAL_TO_FMTSTR(actual_position, 2, TRUE));

LowElevationEvent(	Trigger := Calibrated AND actual_position < 5.0, 
				Level := ADSLOG_MSGTYPE_WARN,
				FormatString := 'Low Elevation: %s',
				OnMessage := LREAL_TO_FMTSTR(actual_position, 2, TRUE));
				
ElevationBrakeEvent( Trigger := NOT enable AND HydraulicsControl.brake_open, 
				Level := ADSLOG_MSGTYPE_WARN,
				FormatString := '%s',
				OnMessage := 'Brake was opened without elevation axis enabled!'); 

TorqueWarning(	
	Trigger := torque_timer.Q, 
	Level := 		ADSLOG_MSGTYPE_WARN,
	FormatString :=	'%s',
	OnMessage := 	'Elevation torque is high.');
	
CalibrationEvent(
	Trigger :=	Calibrated,
	Level :=	ADSLOG_MSGTYPE_HINT,
	OnMessage := 'Elevation is calibrated.'
	);

END_PROGRAM

// ---- POUs/CoverControl.TcPOU
PROGRAM CoverControl
VAR_INPUT
	// resets all drives after an error has occured
	reset:		BOOL;
	// open the cover in proper order
	open:		BOOL;
	// close the cover in proper order
	close:		BOOL;
	// actual active cover in manual mode, 0 for automatic = all covers active
	active_cover:	INT;

END_VAR
VAR_OUTPUT
	// is TRUE, if all covers are open
	isopen:			BOOL;
	// is TRUE, if all covers are closed
	isclosed:		BOOL;
	// is TRUE if any cover-driver reports an error
	Error: 	BOOL;
	// warning state of the DC drives
	Warning: BOOL;
	// cover1 is open
	Cover1_opened, 
	// cover1 is closed
	Cover1_closed:	BOOL;
	// cover2 is open
	Cover2_opened, 
	// cover2 is closed
	Cover2_closed:	BOOL;
	// cover3 is open
	Cover3_opened, 
	// cover3 is closed
	Cover3_closed:	BOOL;
	Cover1_error: BOOL;
	Cover2_error: BOOL;
	Cover3_error: BOOL;
END_VAR
VAR
	// delay timer for opening cover2
	open2_delay: 	TON := (PT:=T#1S);;
	// dely timer for closing cover3
	close3_delay : 	TON := (PT:=T#3S);;
	// trigger for error
	error_trigger:	SR;
	//error event for cover1
	Cover1_Event,
	Cover2_Event,
	Cover3_Event:	FB_EventLog;
	// timeout event for cover1
	Cover1_Timeout_Event,
	Cover2_Timeout_Event,
	Cover3_Timeout_Event:	FB_EventLog;
	// log if covers are open
	Covers_opened_event,
	// log if covers are closed
	Covers_closed_event:	FB_EventLog;
	// Event log for a generic drive error
	Covers_Error_event:		FB_EventLog;
	// Event log for a generic drive warning
	Covers_Warning_event:		FB_EventLog;
END_VAR

(*
This is the control for the two (three) telescope covers. 
The correct order for opening is 1->3->2 and for closing 2->3->1.
GVL Open and close signals are inverted
*)

// close has precedence over open
IF close THEN
	open := FALSE;
END_IF

Cover1_opened := NOT GVL_Telescope.cover1_open;
Cover2_opened := NOT GVL_Telescope.cover2_open;
Cover3_opened := NOT GVL_Telescope.cover3_open;
Cover1_closed := NOT GVL_Telescope.cover1_closed;
Cover2_closed := NOT GVL_Telescope.cover2_closed;
Cover3_closed := NOT GVL_Telescope.cover3_closed;
Cover1_error := Cover1_opened AND Cover1_closed;
Cover2_error := Cover2_opened AND Cover2_closed;
Cover3_error := Cover3_opened AND Cover3_closed;

// wait for cover2 until cover3 has left the closed state
open2_delay(IN := open AND NOT cover3_closed);
// wait for cover3 until cover2 has left the open state
close3_delay(IN := close AND NOT cover2_opened);

IF close THEN
	GVL_Telescope.close_cover1 := GVL_Telescope.cover1_closed AND NOT GVL_Telescope.cover3_closed;
	GVL_Telescope.close_cover2 := GVL_Telescope.cover2_closed;
	GVL_Telescope.close_cover3 := GVL_Telescope.cover3_closed AND close3_delay.Q;
ELSIF open THEN
	GVL_Telescope.open_cover1 := GVL_Telescope.cover1_open;
	GVL_Telescope.open_cover2 := GVL_Telescope.cover2_open AND open2_delay.Q;
	GVL_Telescope.open_cover3 := GVL_Telescope.cover3_open;			
END_IF


// we are open, if all covers are open
isopen := cover3_opened AND cover2_opened AND cover1_opened;
// we are closed, if all covers are closed
isclosed := cover2_closed AND cover3_closed AND cover1_closed;
// error indicates an axis error on any axis
error_trigger(SET1 := Cover1_error OR Cover2_error OR Cover3_error,
				RESET := reset,
				Q1 => error);
//Warning := Cover1_control.Warning OR Cover2_control.Warning OR Cover3_control.Warning;

IF isclosed THEN
	close := FALSE;
END_IF

IF isopen THEN
	open := FALSE;
END_IF

Covers_Error_Event.OnMessage := 'Cover drive error';
IF Error THEN
	IF Cover3_error THEN 
		Covers_Error_Event.OnMessage := 'Cover 3 has a drive error.';
	END_IF
	IF Cover2_error THEN 
		Covers_Error_Event.OnMessage := 'Cover 2 has a drive error.';
	END_IF
	IF Cover1_error  AND NOT GVL_Main.isRoboTel THEN 
		Covers_Error_Event.OnMessage := 'Cover 1 has a drive error.';
	END_IF
END_IF

Covers_Error_event(	Trigger := Error, 
					Level := ADSLOG_MSGTYPE_ERROR);

Covers_Warning_event(	Trigger := Warning, 
						Level := ADSLOG_MSGTYPE_WARN);

// raise an error, if both opened and closed signals are activated
// handle RoboTel differently
Cover1_Event(	Trigger := cover1_opened AND cover1_closed AND NOT GVL_Main.isRoboTel,
				Level := ADSLOG_MSGTYPE_ERROR, 
				OnMessage := 'Cover1: limit switch error');

Cover2_Event(Trigger := cover2_opened AND cover2_closed,
				Level := ADSLOG_MSGTYPE_ERROR, 
				OnMessage := 'Cover2: limit switch error');

Cover3_Event(Trigger := cover3_opened AND cover3_closed,
				Level := ADSLOG_MSGTYPE_ERROR, 
				OnMessage := 'Cover3: limit switch error');

//trigger an event, if we encounter a timeout
// handle RoboTel differently

Cover1_Timeout_Event(Trigger := FALSE,
				Level := ADSLOG_MSGTYPE_ERROR, 
				OnMessage := 'Cover1: Timeout');

Cover2_Timeout_Event(Trigger := FALSE,
				Level := ADSLOG_MSGTYPE_ERROR, 
				OnMessage := 'Cover2: Timeout');

Cover3_Timeout_Event(Trigger := FALSE,
				Level := ADSLOG_MSGTYPE_ERROR, 
				OnMessage := 'Cover3: Timeout');
// Log if we are opened
Covers_opened_event(Trigger := isopen,
					Level := ADSLOG_MSGTYPE_WARN,
					OnMessage := 'All covers are open');
//log if we are closed
Covers_closed_event(Trigger := isclosed,
					Level := ADSLOG_MSGTYPE_HINT,
					OnMessage := 'All covers are closed');

END_PROGRAM

// ---- POUs/Functions/NCError_TO_STRING.TcPOU
FUNCTION NCError_TO_STRING : STRING(255)
VAR_INPUT
	// NC Error ID
	ErrorID:	UDINT;
END_VAR
VAR
END_VAR

NCError_TO_STRING := '';

CASE ErrorID OF
	16#D012:	NCError_TO_STRING := 'Control and power section ready (no error)';
	16#D013:	NCError_TO_STRING := 'Axis in operation (no error)';
	16#4220:	NCError_TO_STRING := 'Group not ready / group not ready for new task';
	16#4253:	NCError_TO_STRING := 'Reference cam became free too soon';
	16#4257:	NCError_TO_STRING := 'Function not allowed';
	16#4260:	NCError_TO_STRING := 'Controller enable';
	16#42EF:	NCError_TO_STRING := 'Axis is locked for motion commands because a stop command is still active';
	16#4466:	NCError_TO_STRING := 'Invalid IO data FOR more than n subsequent NC cycles (encoder)';
	16#4550: 	NCError_TO_STRING := 'Following error monitoring (position)';
	16#4650:	NCError_TO_STRING := 'Drive hardware not ready to operate';
	16#4B07:	NCError_TO_STRING := 'Timeout axis function block';
	16#4B09:	NCError_TO_STRING := 'Axis is not ready';
	16#4B0A:	NCError_TO_STRING := 'Error during referencing';
	16#ECD0:	NCError_TO_STRING := 'Positive limit switch warning.';				
	16#ED43:	NCError_TO_STRING := 'Under-voltage - DC link.';				
	16#F324:	NCError_TO_STRING := 'Excessive position command value deviation';				
	16#F601:	NCError_TO_STRING := 'Calibrate commutation offset error.';				

ELSE
	NCError_TO_STRING := DWORD_TO_HEXSTR(ErrorID, 4, FALSE);
END_CASE

END_FUNCTION

// ---- POUs/FilterWheelControl.TcPOU
PROGRAM FilterWheelControl
VAR_INPUT
	// enable the axis
	Enable:				BOOL;
	// reset the axis(-error)
	Reset:				BOOL;
	// move counter-clockwise
	left:				BOOL;
	// move clockwise
	right:				BOOL;
	// TRUE, if the filter is in position and wheel has come to rest
	Ready:				BOOL;
	// filter position
	filter_position: 	USINT;
	// move to given position
	MoveAxis: 			BOOL;
	// calibrate the axis
	HomeAxis:			BOOL;
END_VAR
VAR_OUTPUT
	// is true if an error occurred
	error: 				BOOL;
	// number of current axis error
	ErrorID:			UDINT;
	act_position:		LREAL;
	// axis has been calibrated
	Calibrated :		BOOL;
END_VAR
VAR
	FilterWheelAxis:	FB_Axis2;
	// axis position to set to with `MoveAxis`
	position:			LREAL;
	// current filter determined from the axis position
	actual_filter:		USINT;
	FilterWheelEvent:	FB_EventLog;
	CalibratedEvent:	FB_EventLog;
	FilterReadyEvent:	FB_Eventlog;
	Calibration1Event:	FB_Eventlog;
	Calibration2Event:	FB_Eventlog;
	
	// last known filter position
	last_filter_position:	USINT;
	HomingMode:			MC_HomingMode := MC_HomingMode.MC_ForceCalibration;
	MQTTTimer : 		TON := (PT:=T#5S);
	CalibrationTrigger1:	R_TRIG;
	CalibrationTrigger2:	F_TRIG;
END_VAR
VAR CONSTANT
	// total number of filters in the filter wheel
	filters:			USINT := 24;
	// current position of the calibration cam. Apply an offset here if necessary
	calibration_position:	LREAL := 1.8;
END_VAR

(* This program controls the filter wheel. 
The current optical filter is selected through `filter_position`.
The number of filters is hard coded to 24.
Position offset: 3285400430
*)

// limit desired filter_position to [0...filters-1]
filter_position := filter_position MOD filters;
// calculate the actual filter position
actual_filter := LREAL_TO_USINT((360.0 - act_position) * filters / 360.0) MOD filters;

Ready := (filter_position = actual_filter) AND (FilterWheelAxis.Standstill OR NOT Enable);
IF Pendantcontrol.telescope_mode = E_TelescopeMode.automatic THEN
	IF FilterWheelAxis.Calibrated THEN
		// if we are on automatic mode then position the filterwheel
		position := MODABS(360.0 - 360.0 * WORD_TO_LREAL(filter_position) / WORD_TO_LREAL(filters), 360.0);
		IF filter_position <> actual_filter THEN
			IF FilterWheelAxis.Ready THEN
				MoveAxis := TRUE;	
			ELSE
				Enable := TRUE;
			END_IF
		END_IF
		IF FilterWheelAxis.MoveDone THEN
			Enable := FALSE;
		END_IF
	ELSE
		IF FilterWheelAxis.Ready THEN
			HomeAxis := TRUE;
		END_IF
	END_IF
END_IF
IF HomeAxis THEN
	IF HomingMode = MC_HomingMode.MC_DefaultHoming THEN
		position := calibration_position;
		filter_position := 0;	
	END_IF
END_IF

Calibrated := FilterWheelAxis.Calibrated;

FilterWheelAxis(
	Enable := 			Enable,
	Reset := 			Reset,
	MoveAxis :=			MoveAxis,
	HomeAxis :=			HomeAxis,
	HomingMode :=		HomingMode,
	Position := 		position, 
	Velocity :=			30.0, //60.0,
	Enable_Positive :=  TRUE,
	Enable_Negative := 	TRUE,
	Jog_Forward :=		left,
	Jog_Backwards := 	right,
	bCalibrationCam :=	NOT GVL_FilterWheel.bCalibrationCam,
	isModuloAxis :=		TRUE,
	ActualPosition => 	act_position,
	Error => 			error,
	ErrorID => 			ErrorID,
	AxisRef :=			GVL_FilterWheel.FilterWheel_AxisRef);

IF FilterWheelAxis.MoveDone THEN
	MoveAxis := FALSE;
END_IF

IF FilterWheelAxis.HomeDone THEN
	HomeAxis := FALSE;
	Enable := FALSE;
END_IF
	
IF FilterWheelAxis.ResetDone THEN
	reset := FALSE;
END_IF

CalibrationTrigger1(CLK := GVL_FilterWheel.bCalibrationCam);
CalibrationTrigger2(CLK := GVL_FilterWheel.bCalibrationCam);


MQTTTimer(IN:=TRUE);
IF actual_filter <> last_filter_position OR MQTTTimer.Q THEN
	MAIN.MQTTClient.Publish('telescope', 'dome', 'FilterPosition', WORD_TO_STRING(actual_filter));
	MAIN.MQTTClient.Publish('telescope', 'dome', 'FilterWheelReady', BOOL_TO_STRING(Ready));
	last_filter_position := actual_filter;
	MQTTTimer(IN:=FALSE);
END_IF

FilterWheelEvent(	
	Trigger := 		Error, 
	Level := 		ADSLOG_MSGTYPE_ERROR,
	FormatString :=	'Filter Wheel Axis Error: %s',
	OnMessage := 	NCError_TO_STRING(ErrorID),
	OffMEssage := 	'OK',
	OffLevel := 	ADSLOG_MSGTYPE_HINT);
	
CalibratedEvent(
	Trigger :=		Calibrated,
	Level := 		ADSLOG_MSGTYPE_HINT,
	FormatString :=	'%s',
	OnMessage := 	'Filter wheel is calibrated.');
	
FilterReadyEvent(
	Trigger :=		(filter_position = actual_filter) AND Calibrated,
	Level := 		ADSLOG_MSGTYPE_HINT,
	FormatString :=	'Filter position %s is ready.',
	OnMessage := 	WORD_TO_STRING(actual_filter));
	
Calibration1Event(
	Trigger :=	CalibrationTrigger1.Q,
	Level := 		ADSLOG_MSGTYPE_HINT,
	FormatString :=	'Calibration raising signal triggered at position: %s',
	OnMessage := 	LREAL_TO_STRING(act_position));

Calibration2Event(
	Trigger :=	CalibrationTrigger2.Q,
	Level := 		ADSLOG_MSGTYPE_HINT,
	FormatString :=	'Calibration falling signal triggered at position: %s',
	OnMessage := 	LREAL_TO_STRING(act_position));

END_PROGRAM

// ---- POUs/FocusControl.TcPOU
PROGRAM FocusControl
VAR_INPUT
	// enable the axis
	enable: BOOL;
	// Move M2 closer to M1
	inward: 	BOOL;
	// Move M2 away from M1
	outward: 	BOOL;	
	// reset the axis(-error)
	reset: 		BOOL;
	// move the axis to new position
	MoveAxis:	BOOL;
	// calibrate the focus axis
	HomeAxis:	BOOL;
	// focus position in millimeters
	position: 		LREAL;
END_VAR

VAR_OUTPUT
	// true if absolute calibration
	Calibrated:	BOOL;
	// true if error
	Error: 		BOOL;
	// ID of NC axis error
	ErrorID:	UDINT;
	// ready signal = drive ready + standstill
	Ready:	BOOL;
END_VAR

VAR
	FocusDelay:			TON;
	BrakeDelay:			TON;
	FocusAxis:			FB_Axis2;
	actual_position:	LREAL;
	// manual override to unlock the focus
	FocusUnlock:		BOOL;
	FocusUnlocked:		BOOL;
	MQTTTimer : 		TON := (PT:=T#5S);
	//getlastposition:	BOOL := TRUE;
	FocusAxisEvent:		FB_EventLog;
	CalibrationEvent:	FB_EventLog;
	HomingMode: 		MC_HOMINGMODE := 		MC_DefaultHoming;
	SetPosition:		MC_SetPosition;
END_VAR

VAR CONSTANT
	// reference position for homing
	homing_position:		LREAL := 92.8936; // 106.5936 - 13.7000
	tolerance:				LREAL := 0.005;
END_VAR
VAR PERSISTENT
	last_position:		LREAL := -1.0;
END_VAR

(*
Focus Control Unit
spindle gear: 5mm
brake: 86 61103H00 Var. 0005 Index C; 24VDC geglattet 0,25 A P1672/R7
motor: Faulhaber ; Schönaich ; 3557K024CR; 454  431 ; Made in germany ==> 5300 rpm
gear: Faulhaber ; MINIMOTOR SA ; swiss made ; 38/1S  43:1 ; 033896  503
Focus is locked by default
70,8W; 0,100A no load current; 2,0 Terminal resistance; 1,950A max Current 
*)
position := LIMIT(5.0, position, 95.0);

GVL_Telescope.focus_unlock := FocusUnlock OR enable;

// wait until the focus is unlocked for n milliseconds
FocusDelay(IN := GVL_Telescope.focus_unlock, PT := T#500MS, Q => FocusUnlocked);
// wait for brake until we are at rest
BrakeDelay(IN := NOT FocusAxis.Busy AND FocusAxis.StandStill, PT := T#4000MS);

// if we are on automatic mode then position the filterwheel
IF Pendantcontrol.telescope_mode = E_TelescopeMode.automatic AND NOT FocusUnlock THEN
	IF FocusAxis.Calibrated THEN
		IF ABS(position - actual_position) > tolerance THEN
			IF FocusAxis.Ready THEN
				MoveAxis := TRUE;
			ELSE
				Enable := TRUE;
			END_IF
		END_IF
		// disable the drive and lock the brake, if we stand for more than n seconds
		IF BrakeDelay.Q THEN
			Enable := FALSE;
		END_IF
		// store actual position, if we are calibrated and locked
		IF NOT GVL_Telescope.focus_unlock THEN
			last_position := actual_position;
		END_IF
	ELSE // not calibrated
		IF FocusAxis.Ready THEN
			HomeAxis := TRUE;
		END_IF
	END_IF
END_IF

IF HomeAxis THEN
	IF last_position > 0.0 THEN
		HomingMode := MC_ForceCalibration; // MC_Direct
		position := last_position;
		SetPosition.Execute := TRUE;
	ELSE
		HomingMode := MC_DefaultHoming;
		position := homing_position;
		SetPosition.Execute := FALSE;
	END_IF
ELSE
	SetPosition.Execute := FALSE;	
END_IF

// deactivate limit switches on homing
MC_SetAcceptBlockedDriveSignal(
	Axis := GVL_Telescope.FocusAxisRef, 
	Enable := HomeAxis);
SetPosition(
	Axis := GVL_Telescope.FocusAxisRef, 
	Position := last_position);
	
	
FocusAxis(	
	Enable := 			FocusUnlocked,
	Reset := 			reset,
	MoveAxis := 		MoveAxis AND FocusUnlocked,
	HomeAxis :=			HomeAxis AND FocusUnlocked,
	HomingMode :=		HomingMode,
	Position := 		position,
	Velocity :=			1.0,
	Enable_Positive := 	NOT GVL_Telescope.focus_limit_far OR HomeAxis,
	Enable_Negative := 	NOT GVL_Telescope.focus_limit_near,
	Jog_Forward :=		outward AND FocusUnlocked,
	Jog_Backwards := 	inward AND FocusUnlocked,
	bCalibrationCam :=  GVL_Telescope.focus_limit_far,
	ActualPosition => 	actual_position,
	Error =>			error,
	ErrorID =>			ErrorID,
	AxisRef :=			GVL_Telescope.FocusAxisRef);	

IF FocusAxis.MoveDone THEN
	MoveAxis := FALSE;
END_IF

IF FocusAxis.HomeDone THEN
	HomeAxis := FALSE;
	Enable := FALSE;
	last_position := position;
END_IF
	
IF FocusAxis.ResetDone THEN
	reset := FALSE;
END_IF

IF FocusAxis.Calibrated OR Error THEN
	HomeAxis := FALSE;
END_IF

IF Error THEN
	last_position := -1.0;
	//FocusAxis.Calibrated := FALSE;
	Calibrated := FALSE;
END_IF

Calibrated := FocusAxis.Calibrated;

Ready := FocusAxis.Ready AND FocusAxis.StandStill OR NOT GVL_Telescope.focus_unlock;

MQTTTimer(IN:=TRUE);
IF MQTTTimer.Q THEN // publish new payload every second
	MQTTTimer(IN:=FALSE);
	MAIN.MQTTClient.Publish('telescope', 'dome', 'FocusPosition', LREAL_TO_FMTSTR(actual_position, 5, TRUE));
	MAIN.MQTTClient.Publish('telescope', 'dome', 'FocusCalibrated', BOOL_TO_STRING(Calibrated));	
	MAIN.MQTTClient.Publish('telescope', 'dome', 'FocusReady', BOOL_TO_STRING(Ready));	
END_IF

FocusAxisEvent(	
	Trigger := 		FocusAxis.Error, 
	Level := 		ADSLOG_MSGTYPE_ERROR,
	FormatString :=	'Focus Axis Error: %s',
	OnMessage := 	NCError_TO_STRING(ErrorID),
	OffMEssage := 	'OK',
	OffLevel := 	ADSLOG_MSGTYPE_HINT);

CalibrationEvent(
	Trigger :=	Calibrated,
	Level :=	ADSLOG_MSGTYPE_HINT,
	OnMessage := 'Focus is calibrated.'
	);

END_PROGRAM

// ---- POUs/DerotatorControl.TcPOU
PROGRAM DerotatorControl
VAR_INPUT
	// enable the derotator
	enable:		BOOL;
	// reset an error
	reset:		BOOL;
	// decrease derotator angle
	left:		BOOL;
	// increase derotator angle
	right:		BOOL;
	// set the absolute position
	position:	LREAL;
	// derotator velocity
	Velocity:	LREAL := 10.0;
	// move to given position
	MoveAxis: 	BOOL;
	// calibrate the axis
	HomeAxis:	BOOL;
	// tracking flag
	Tracking:	BOOL;
	// stop the Axis
	StopAxis:	BOOL;
	// diagnostic error code reset
	bSoEReset: 			BOOL;
END_VAR
VAR_OUTPUT
	// error flag
	Error:				BOOL;
	// nc error id
	ErrorID:			UDINT;
	// actual position of the derotator
	actual_position:	LREAL;
	// calibrated flag
	Calibrated:			BOOL;
	// axis ready flag
	Ready:				BOOL;
	// position to move the axis to
	slewtime: 			LREAL;
END_VAR
VAR
	// trigger for the torque error
	TorqueError:		TON := (PT := T#3S);
	// axis function block
	DerotatorAxis:		FB_Axis2;
	
	DerotatorEvent:		FB_EventLog;
	// torque warning event
	TorqueWarning:		FB_EventLog;
	// torque calibration event
	CalibrationEvent:	FB_EventLog;
	// diagnostic low-level event
	DerotatorDiagnosticEvent: FB_EventLog;
	// percentage of the derotator torque
	derotator_torque:	REAL;
	// read slewtime
	ReadParameter:		MC_ReadParameter;
	fbSoEReset: 		FB_SoEReset;
	DiagnosticError:	BOOL;
END_VAR
VAR CONSTANT
	// current position of the calibration cam. Apply an offset here if necessary
	calibration_position:	LREAL := 438.4623; // calibration in positive direction (was 460.0)
END_VAR

(*
Selection 6
Homing in Endlage:

https://infosys.beckhoff.com/index.php?content=../content/1031/ax5000_usermanual/html/ax5000_homing_hardware_end_position.htm&id=12221
NC-Interface:
PlcToNc-Achsinterface, Bit 8 namens AcceptBlockedDriveSignal im nDeCtrlDWord

SPS-Interface:
TcNc-Lib, siehe SPS-Funktion AxisSetAcceptBlockedDriveSignal in der TwinCAT  PLC Library: NC.
*)

position := LIMIT(-70, position, 380);

IF enable AND NOT DerotatorAxis.Calibrated THEN
	HomeAxis := TRUE;
END_IF

IF DerotatorAxis.Calibrated THEN
	HomeAxis := FALSE;
	Calibrated := DerotatorAxis.Calibrated;
END_IF
	
IF HomeAxis THEN
	position := calibration_position;
END_IF

DeRotatorAxis(
	enable := 			enable,
	Reset := 			Reset,
	MoveAxis :=			MoveAxis,
	HomeAxis :=			HomeAxis,
	StopAxis :=			StopAxis,
	HomingMode :=		MC_ForceCalibration,
	Position := 		position, 
	Velocity :=			Velocity,
	Enable_Positive := 	NOT GVL_Telescope.Derotator_inputs.0,
	Enable_Negative := 	NOT GVL_Telescope.Derotator_inputs.1,
	Jog_Forward := 		right,
	Jog_Backwards := 	left,
	bCalibrationCam :=	GVL_Telescope.Derotator_inputs.0,
	isModuloAxis :=		FALSE,
	Tracking :=			Tracking,
	ActualPosition => 	actual_position,
	Error => 			Error,
	ErrorID => 			ErrorID,
	AxisRef :=			GVL_Telescope.DerotatorAxisRef);
	
IF DeRotatorAxis.MoveDone OR Reset OR Error THEN
	MoveAxis := FALSE;
END_IF

IF DeRotatorAxis.HomeDone OR Reset OR Error THEN
	HomeAxis := FALSE;
END_IF
	
IF DeRotatorAxis.ResetDone THEN
	reset := FALSE;
END_IF

IF DeRotatorAxis.StopDone THEN
	StopAxis := FALSE;
END_IF

DiagnosticError := FALSE;
IF GVL_Telescope.Derotator_diagnostic < 16#D012 AND GVL_Telescope.Derotator_diagnostic > 16#D014 THEN
	DiagnosticError := TRUE;
	ErrorID := GVL_Telescope.Derotator_diagnostic;
	bSoeReset := reset;
END_IF

Ready := DeRotatorAxis.Ready;

ReadParameter(	Axis := GVL_Telescope.DerotatorAxisRef, 
				Enable := DeRotatorAxis.InMotion, 
				ParameterNumber := MC_AxisParameter.AxisRemainingTimeToGo, 
				ReadMode := E_ReadMode.READMODE_CYCLIC);
				
IF ReadParameter.Valid THEN
	slewtime := ReadParameter.Value;
END_IF

IF bSoEReset THEN
	fbSoEReset(
		Axis := GVL_Telescope.DerotatorAxisRef,
		Execute := TRUE,
		Timeout := DEFAULT_ADS_TIMEOUT);
 	IF NOT fbSoEReset.Busy THEN
		fbSoEReset(Axis := GVL_Telescope.DerotatorAxisRef, Execute := FALSE);
		bSoEReset := FALSE;
		Reset := TRUE;
	END_IF
END_IF

derotator_torque := GVL_Telescope.Derotator_torque / 10.0;
// nominal torque is 3%, max is 25%
TorqueError(IN := ABS(derotator_torque) > 20.0);

DerotatorEvent(	
	Trigger := 		Error, 
	Level := 		ADSLOG_MSGTYPE_ERROR,
	FormatString :=	'Derotator Axis Error: %s',
	OnMessage := 	NCError_TO_STRING(ErrorID),
	OffMEssage := 	'OK',
	OffLevel := 	ADSLOG_MSGTYPE_HINT);
	
DerotatorDiagnosticEvent(	
	Trigger := 		DiagnosticError, 
	Level := 		ADSLOG_MSGTYPE_ERROR,
	FormatString :=	'Derotator Axis Diagnostic Error: %s',
	OnMessage := 	NCError_TO_STRING(GVL_Telescope.Derotator_diagnostic));
	
TorqueWarning(	
	Trigger := 		TorqueError.Q, 
	Level := 		ADSLOG_MSGTYPE_WARN,
	FormatString :=	'%s',
	OnMessage := 	'Derotator torque is high.');

CalibrationEvent(	
	Trigger := 		Calibrated, 
	Level := 		ADSLOG_MSGTYPE_HINT,
	OnMessage := 	'Derotator is calibrated.');

END_PROGRAM

// ---- POUs/Functions/F_DerotatorPosition2.TcPOU
FUNCTION F_DerotatorPosition2 : LREAL
VAR_INPUT
	// azimuth of the target
	azimuth: LREAL;
	// elevation of the target in degrees
	elevation: LREAL;
	// declination of the target in degrees
	declination: LREAL;
	// latitude in degrees
	latitude:	LREAL;
	// sign for elevation
	sign:	LREAL := 1.0;
END_VAR
VAR
	// parallactic angle
	de, az, el, la: LREAL;
	parallactic_angle:	LREAL;
	//zenith_distance: LREAL;
END_VAR
VAR CONSTANT
	d2r:	LREAL := PI/180.0;
	r2d:	LREAL := 180.0/PI;
	//h2r:	LREAL := PI/12.0;
	//h2d:	LREAL := 15.0;
END_VAR

// calculate the parallactic angle
de := LIMIT(-90.0, declination, 90.0) * d2r;
az := MODABS(azimuth, 360.0) * d2r;
el := LIMIT(0.0, elevation, 90.0) * d2r;
la := LIMIT(-90.0, latitude, 90.0) * d2r;

parallactic_angle := - r2d * ATAN2(SIN(az), TAN(la)*COS(el)-SIN(el)*COS(az));

F_DerotatorPosition2 := parallactic_angle - sign * elevation;
IF F_DerotatorPosition2 <= -70.0 OR F_DerotatorPosition2 >= 380.0 THEN
	F_DerotatorPosition2 := MODABS(F_DerotatorPosition2, 360.0);
END_IF

END_FUNCTION

// ---- POUs/Functions/F_Elevationvelocity.TcPOU
FUNCTION F_Elevationvelocity : LREAL
VAR_INPUT
	// azimuth in degrees
	azimuth:	LREAL;
	// observers latitude in degrees
	latitude:	LREAL;
END_VAR
VAR
END_VAR
VAR CONSTANT
	// Earth's angular rotation frequency in [deg/s]
	Omega: LREAL := 4.178074605556E-3;
	d2r:	LREAL := PI/180.0;
	//r2d:	LREAL := 180.0/PI;
END_VAR

//returns the rotational velocity for the azimuth in degrees per second
F_Elevationvelocity := SIN(azimuth*d2r) * COS(latitude*d2r) * Omega;

END_FUNCTION

// ---- POUs/Functions/F_Azimuthvelocity.TcPOU
FUNCTION F_Azimuthvelocity : LREAL
VAR_INPUT
	// elevation in degrees
	elevation: 	LREAL;
	// azimuth in degrees
	azimuth:	LREAL;
	// observers latitude in degrees
	latitude:	LREAL;
END_VAR
VAR
END_VAR
VAR CONSTANT
	// Earth's angular rotation frequency in [deg/s]
	Omega: LREAL := 4.178074605556E-3;
	d2r:	LREAL := PI/180.0;
	//r2d:	LREAL := 180.0/PI;
END_VAR

IF ABS(COS(elevation * d2r))> 1.0e-3 THEN
	F_Azimuthvelocity := (SIN(latitude * d2r) - COS(latitude * d2r) * COS(azimuth * d2r) * TAN(elevation *d2r))* Omega;
ELSE
	F_Azimuthvelocity := 0.0;	
END_IF

END_FUNCTION

// ---- POUs/Transformer.TcPOU
PROGRAM Transformer
VAR_INPUT
	// reset signal for the error condition
	reset_error:		BOOL := FALSE;
	// signal to start the transformer
	softstart_trafo:	BOOL;
END_VAR
VAR_OUTPUT
	// indicates the phases for the hydraulics
	phase_available:	BOOL;
	// trafo failed to start after timeout
	power_failure:		BOOL;
	// restart was inhibited
	restart_inhibited:	BOOL;
END_VAR
VAR
	// watchdog for trafo softstarter
	power_watchdog: 	TON;
	// timer to measure the startup time
	power_timer:		FB_timer;
	// timeout for the startup
	startup_timeout:	TIME := T#5S;
	// error state
	power_error_state:	SR;
	// restart inhibitor
	restart_inhibit:	TOF;
	PowerEvent:			FB_EventLog;
	PowerLog:			FB_EventLog;
	
END_VAR

power_timer(bStart := GVL_Main.softstart_trafo, bStop := power_OK);
power_watchdog(IN := GVL_Main.softstart_trafo AND NOT power_OK,
				PT := startup_timeout,
				Q => power_failure);
power_error_state(SET1 := power_failure, RESET := reset_error);
restart_inhibit(IN := GVL_MAIN.trafo_bypassed, PT := T#5S);

restart_inhibited := NOT GVL_MAIN.trafo_bypassed AND restart_inhibit.Q;
IF restart_inhibited THEN
	softstart_trafo := FALSE;
END_IF
GVL_Main.softstart_trafo := softstart_trafo AND NOT error;

	
phase_available := PowerMonitoring.phaseOK;

PowerEvent(	
	Trigger := 		power_failure, 
	Level := 		ADSLOG_MSGTYPE_ERROR,
	FormatString :=	'%s',
	OnMessage := 	'Servo power FAILURE!',
	OffMEssage := 	'Servo power OK');
PowerLog(	
	Trigger := 		power_OK, 
	Level := 		ADSLOG_MSGTYPE_HINT,
	FormatString :=	'%s',
	OnMessage := 	'Mains power is ON',
	OffMEssage := 	'Mains power is OFF');

PROPERTY error : BOOL
GET
error := power_error_state.Q1;
END_GET
END_PROPERTY

PROPERTY power_ok : BOOL
// indicates the power state for the AX5000
GET
power_ok := GVL_main.trafo_bypassed;
END_GET
END_PROPERTY

METHOD reset : BOOL
VAR_INPUT
END_VAR
IF error THEN
	reset_error := TRUE;
ELSE
	reset_error := FALSE;
END_IF
END_METHOD

METHOD start : BOOL
VAR_INPUT
END_VAR
softstart_trafo := TRUE;
END_METHOD

PROPERTY startup_time : TIME
GET
startup_time := power_timer.tDifference;
END_GET
SET
startup_timeout := startup_time;
END_SET
END_PROPERTY

METHOD stop : BOOL
VAR_INPUT
END_VAR
softstart_trafo := FALSE;
END_METHOD

END_PROGRAM

// ---- POUs/FunctionBlocks/FB_Timer.TcPOU
FUNCTION_BLOCK FB_Timer
VAR_INPUT
	bStart          : BOOL := FALSE;
	bStop			: BOOL := FALSE;
END_VAR
VAR_OUTPUT
    tDifference     : TIME;
END_VAR
VAR
    StartTrigger,
	StopTrigger		: R_TRIG;
    StartTime    	: TIME;
    StopTime    	: TIME;
END_VAR

(*
Timer functionblock

Source:
https://infosys.beckhoff.de/index.php?content=../content/1031/tc3_plc_intro/2529365899.html&id=
*)
StartTrigger(CLK := bStart);
StopTrigger(CLK := bStop);

IF StartTrigger.Q THEN
    StartTime  := TIME();
END_IF

IF StopTrigger.Q THEN
    StopTime  := TIME();
    tDifference   := StopTime - StartTime;    // The difference will be T#5s
END_IF

END_FUNCTION_BLOCK

// ---- POUs/PowerMonitoring.TcPOU
PROGRAM PowerMonitoring
VAR_INPUT
END_VAR
VAR_OUTPUT
	phaseOK:				BOOL;
END_VAR
VAR
	Overvoltage				AT%I*: BOOL;
	Overcurrent				AT%I*: BOOL;
	VoltageGuardWarning		AT%I*: BOOL;
	VoltageGuardError		AT%I*: BOOL;
	CurrentGuardWarning		AT%I*: BOOL;
	CurrentGuardError		AT%I*: BOOL;
	NeutralCurrentGuardWarning		AT%I*: BOOL;
	NeutralCurrentGuardError		AT%I*: BOOL;
	Voltage					AT%I*: REAL;
	Current					AT%I*: REAL;
	ActivePower				AT%I*: REAL;
	ApparentPower			AT%I*: REAL;
	ReactivePower			AT%I*: REAL;
	PowerQualityFactor		AT%I*: REAL;
	Frequency				AT%I*: REAL;
	PowerFactor				AT%I*: REAL;
	NeutralLineCurrent		AT%I*: REAL;
	L1L2Voltage				AT%I*: REAL;
	L2L3Voltage				AT%I*: REAL;
	L3L1Voltage				AT%I*: REAL;
	MQTTTimer: 				TON := (PT:=T#10S);
	PowerWarningDelay:		TON := (PT:=T#100MS);
	PowerWarningRetain:		TOF := (PT:=T#2000MS);
	
	PowerError:				FB_EventLog;
	PowerWarning:			FB_EventLog;
	NeutralCurrentEvent:			FB_EventLog;
END_VAR

phaseOK := L1L2Voltage > 360.0 AND L2L3Voltage > 360.0 AND L3L1Voltage > 360.0;

IF NeutralCurrentGuardError THEN
	NeutralCurrentEvent.Trigger := TRUE;
	NeutralCurrentEvent.OnMessage := 	'Neutral Line Current ERROR!';
	NeutralCurrentEvent.Level := ADSLOG_MSGTYPE_ERROR;
ELSIF NeutralCurrentGuardWarning THEN
	NeutralCurrentEvent.Trigger := TRUE;
	NeutralCurrentEvent.OnMessage := 	'Neutral Line Current WARNING!';
	NeutralCurrentEvent.Level := ADSLOG_MSGTYPE_WARN;
ELSE
	NeutralCurrentEvent.Trigger := FALSE;
END_IF

PowerWarningDelay(IN := VoltageGuardWarning OR CurrentGuardWarning);
PowerWarningRetain(IN := PowerWarningDelay.Q);

// MQTT Section
MQTTTimer(IN:=TRUE);
IF MQTTTimer.Q OR VoltageGuardWarning OR CurrentGuardWarning THEN // publish new payload every second
	MQTTTimer(IN:=FALSE);

	MAIN.MQTTClient.Publish('telescope', 'power', 'Overvoltege',	BOOL_TO_STRING(Overvoltage));
	MAIN.MQTTClient.Publish('telescope', 'power', 'Overcurrent',	BOOL_TO_STRING(Overcurrent));

	MAIN.MQTTClient.Publish('telescope', 'power', 'VoltageGuardWarning',	BOOL_TO_STRING(VoltageGuardWarning));
	MAIN.MQTTClient.Publish('telescope', 'power', 'VoltageGuardError',		BOOL_TO_STRING(VoltageGuardError));
	MAIN.MQTTClient.Publish('telescope', 'power', 'CurrentGuardWarning',	BOOL_TO_STRING(CurrentGuardWarning));
	MAIN.MQTTClient.Publish('telescope', 'power', 'CurrentGuardError',		BOOL_TO_STRING(CurrentGuardError));

	MAIN.MQTTClient.Publish('telescope', 'power', 'Voltage', 		REAL_TO_STRING(Voltage));
	MAIN.MQTTClient.Publish('telescope', 'power', 'Current',		REAL_TO_STRING(Current));
	MAIN.MQTTClient.Publish('telescope', 'power', 'ActivePower',	REAL_TO_STRING(ActivePower));
	MAIN.MQTTClient.Publish('telescope', 'power', 'ApparentPower',	REAL_TO_STRING(ApparentPower));
	MAIN.MQTTClient.Publish('telescope', 'power', 'ReactivePower',	REAL_TO_STRING(ReactivePower));
	MAIN.MQTTClient.Publish('telescope', 'power', 'PowerQualityFactor',	REAL_TO_STRING(PowerQualityFactor));
	MAIN.MQTTClient.Publish('telescope', 'power', 'Frequency',		REAL_TO_STRING(Frequency));
	MAIN.MQTTClient.Publish('telescope', 'power', 'PowerFactor',	REAL_TO_STRING(PowerFactor));
	MAIN.MQTTClient.Publish('telescope', 'power', 'NeutralLineCurrent',	REAL_TO_STRING(NeutralLineCurrent));

	MAIN.MQTTClient.Publish('telescope', 'power', 'L1L2Voltage',	REAL_TO_STRING(L1L2Voltage));
	MAIN.MQTTClient.Publish('telescope', 'power', 'L2L3Voltage',	REAL_TO_STRING(L2L3Voltage));
	MAIN.MQTTClient.Publish('telescope', 'power', 'L3L1Voltage',	REAL_TO_STRING(L3L1Voltage));	
END_IF

// EventLog section
PowerError(	
	Trigger := 		VoltageGuardError OR CurrentGuardError, 
	Level := 		ADSLOG_MSGTYPE_ERROR,
	FormatString :=	'%s',
	OnMessage := 	'electrical power:	ERROR!');
	
PowerWarning(	
	Trigger := 		PowerWarningRetain.Q, 
	Level := 		ADSLOG_MSGTYPE_WARN,
	FormatString :=	'%s',
	OnMessage := 	'electrical power:	WARNING!');

NeutralCurrentEvent(
	FormatString :=	'%s',
	OnMessage := 	'electrical power:	WARNING!');

END_PROGRAM

// ---- POUs/FunctionBlocks/FB_EQ2HOR.TcPOU
FUNCTION_BLOCK FB_EQ2HOR
VAR_INPUT
	RA: 		LREAL;	// Right Ascension of object  (J2000) in degrees (FK5)
	Dec: 		LREAL;	// Declination of object (J2000) in degrees (FK5)
	JD: 		LREAL;	// Julian Date
	LAT: 		LREAL;	// north geodetic latitude of location in degrees
	LON: 		LREAL; 	// EAST longitude of location in degrees (Specify west longitude with a negative sign.)
	ALTITUDE:	LREAL := 0.0;  // The altitude of the observing location, in meters. [default=0].  
	WS:			BOOL := FALSE; //  Set this to TRUE get the azimuth measured westward FROM south (NOT East of North).
	PRECESS:	BOOL := TRUE; // Set this to 1 to force precession [default], 0 for no precession correction
	NUTATE:		BOOL := TRUE; // Set this to 1 to force nutation [default], 0 for no nutation.
	ABERRATION:	BOOL := TRUE; // Set this to 1 to force aberration correction [default], 0 for no correction.
	REFRACT:	BOOL := TRUE; // Set to 1 to force refraction correction [default], 0 for no correction.
END_VAR
VAR_OUTPUT
	alt: 	LREAL; // altitude (in degrees)
	az:		LREAL; // azimuth angle (in degrees, measured EAST FROM NORTH, but see keyword WS above.)
	ha:		LREAL; // hour angle (in degrees) (optional)	
END_VAR
VAR
	ra_, dec_, tstart, J_now: LREAL;
	s_now: STRING;
	fbprecess: FB_PRECESS;
	lmst: LREAL;
	last: LREAL;
	d_psi: LREAL;
	eps: LREAL;
	hadec2altaz:	FB_HADEC2ALTAZ;
	co_nutate: 		FB_CO_NUTATE;
	co_aberration:	CO_ABERRATION;
	co_refract:		CO_REFRACT;
	dra1, dra2: LREAL;
	ddec1, ddec2 : LREAL;
END_VAR
VAR CONSTANT
	d2r:	LREAL := PI/180.0;
	h2r:	LREAL := PI/12.0;
	h2d:	LREAL := 15.0;
END_VAR

(* source https://idlastro.gsfc.nasa.gov/ftp/pro/astro/eq2hor.pro 

PURPOSE:
	Convert celestial  (ra-dec) coords to local horizon coords (alt-az).

DESCRIPTION:
This  code calculates horizon (alt,az) coordinates from equatorial
(ra,dec) coords.   It is typically accurate to about 1 arcsecond or better (I
have checked the output against the publicly available XEPHEM software). It
performs precession, nutation, aberration, and refraction corrections.  The
perhaps best thing about it is that it can take arrays as inputs, in all
variables and keywords EXCEPT Lat, lon, and Altitude (the code assumes these
aren't changing), and uses vector arithmetic in every calculation except
when calculating the precession matrices.
*)

ra_ := ra;
dec_ := dec;

tstart := 2000.0;

(* ******************************************************************************
 PRECESS coordinates to current date
 (uses astro lib procedure PRECESS.pro)
*)
J_now := (JD - 2451545.0)/365.25 + 2000.0; // compute current equinox
IF precess THEN
	fbprecess( ra := ra_, dec := dec_, 
	EQUINOX1 := tstart, EQUINOX2 := J_now, 
	ra_precessed =>ra_, dec_precessed => dec_);
END_IF

(******************************************************************************
 calculate NUTATION and ABERRATION Corrections to Ra-Dec 
*)

IF NUTATE THEN
	co_nutate(	jd := jd, 
				ra := ra_, 
				dec := dec_, 
				d_ra => dra1, 
				d_dec => ddec1, 
				eps=>eps, 
				d_psi=>d_psi);
	ra_ := ra_ + dra1/3600.0;
	dec_ := dec_ + ddec1/3600.0;
END_IF

IF ABERRATION THEN	
	co_aberration(	jd := jd, 
					ra := ra_, 
					dec := dec_, 
					d_ra => dra2, 
					d_dec => ddec2, 
					eps := eps);
	ra_ := ra_ + dra2/3600.0;
	dec_ := dec_ + ddec2/3600.0;
END_IF

(***************************************************************************************
Calculate LOCAL MEAN SIDEREAL TIME *)
lmst := ct2lst(lon, jd);  // get LST (in hours) - note:this is independent of time zone  since giving jd
lmst := lmst*h2d ; //convert LMST to degrees (btw, this is the RA of the zenith)
// calculate local APPARENT sidereal time
last := lmst + d_psi *COS(eps*d2r)/3600.0 ; //add correction in degrees

(******************************************************************************
 Find hour angle (in DEGREES) *)
ha := last - ra_;
ha := MODABS(ha, 360.0);

(*******************************************************************************
 Now do the spherical trig to get APPARENT alt,az. *)
hadec2altaz(	ha := ha, 
				dec := dec_, 
				lat := lat, 
				alt => alt, 
				az => az, 
				WS := WS);

(********************************************************************************************
 Make Correction for ATMOSPHERIC REFRACTION
 (use this for visible and radio wavelengths; author is unsure about other wavelengths.
  See the comments in CO_REFRACT for more details.) *)
IF refract THEN 
	co_refract(	old_alt := alt, 
				altitude := altitude, 
				to_observed := TRUE, 
				new_alt => alt);
END_IF

END_FUNCTION_BLOCK

// ---- POUs/FunctionBlocks/FB_HOR2EQ2.TcPOU
FUNCTION_BLOCK FB_HOR2EQ2
VAR_INPUT
	//altitude (in degrees)
	alt: 		LREAL;  
	//azimuth angle (in degrees, measured EAST from NORTH, but see keyword WS below.) [scalar or vector]
	az:			LREAL;
	// Julian Date [scalar or vector], double precision
	JD: 		LREAL;
	// observers latitude (degrees)
	lat:		LREAL;
	// observers longitude (degrees)
	lon:		LREAL;
	// observers altitude (unused)
	altitude:	LREAL := 0.0;
END_VAR
VAR_OUTPUT
	// Right Ascension of object  (J2000) in degrees (FK5)
	ra: 	LREAL;
	// Declination of object (J2000) in degrees (FK5)
	dec:	LREAL;
	// hour angle (in degrees)
	ha:		LREAL;
END_VAR
VAR
	alt_rad, lat_rad:	LREAL;
	az_rad:		LREAL;
	dec_rad:	LREAL;
	cosha, sinha, sindec:	LREAL;
	lst: 	LREAL;
END_VAR
VAR CONSTANT
	d2r:	LREAL := PI/180.0;
	r2d:	LREAL := 180.0/PI;
	//h2r:	LREAL := PI/12.0;
	h2d:	LREAL := 15.0;
END_VAR

alt_rad := alt * d2r;
lat_rad := lat * d2r;
az_rad := az * d2r;
// sin(dec) = sin(alt)*sin(phi) + cos(alt)*cos(phi)*cos(az)
sindec := SIN(alt_rad)*SIN(lat_rad) + COS(alt_rad)*COS(lat_rad)*COS(az_rad);
dec_rad := ASIN(sindec);
dec := dec_rad * r2d;
//sin(ha) = -sin(azimuth)*cos(altitude)/cos(dec)
IF ABS( COS(dec_rad)) > 0.0 THEN
	sinha := -SIN(az_rad) * COS(alt_rad) / COS(dec_rad);
ELSE
	sinha := 0.0;
END_IF
// cos(ha) = (sin(alt) - sin(dec)*sin(phi))/(cos(dec)*cos(phi))
IF ABS(COS(dec_rad) * COS(lat_rad)) > 0.0 THEN
	cosha := (SIN(alt_rad) - SIN(dec_rad)*SIN(lat_rad)) / (COS(dec_rad) * COS(lat_rad));
ELSE
	cosha := 0.0;
END_IF

// tan(ha) = sin(ha)/cos(ha)
ha := ATAN2(sinha, cosha) * r2d;
ha := MODABS(ha, 360.0);
// ra = t - ha
lst := ct2lst(lon, jd) * 15.0;
ra := lst - ha;
ra := MODABS(ra, 360.0);

END_FUNCTION_BLOCK

// ---- POUs/FunctionBlocks/FB_LightTimer.TcPOU
FUNCTION_BLOCK FB_LightTimer
VAR_INPUT
	IN: BOOL;
	PT: TIME := T#60S;
END_VAR
VAR_OUTPUT
	Q: BOOL;
END_VAR
VAR
	SR1 : SR;
	rtrig: R_TRIG;
	ton1 : TON;
END_VAR

(*
This is a simple light control based on a impulse switch.
The output Q goes high on the rising edge of the input IN.
The output Q stays high until the time PT runs out or another rising edge on IN is detected.
*)

// detect the rsing edge of the input
rtrig(CLK := IN);
// reset the input after PT time
ton1(IN := Q,
		PT := PT);
// sets the flip-flop on the first rising edge, reset it on the second rising edge or when time is up.
SR1(SET1 := rtrig.Q AND NOT Q,
	RESET := ton1.Q OR (Q AND rtrig.Q),
	Q1 => Q);

END_FUNCTION_BLOCK

// ---- POUs/FunctionBlocks/FB_TimeAverage.TcPOU
FUNCTION_BLOCK FB_TimeAverage
VAR_INPUT
	IN:		REAL;
	PT:		TIME := T#4400MS;
END_VAR
VAR_OUTPUT
	AVG:	REAL;
	MINAVG:	REAL;
	MAXAVG:	REAL;
	Overflow: BOOL;
END_VAR
VAR
	fbCycle	:TON;
	buffer:	ARRAY[0..30000] OF REAL;
	index:	INT := 0;
	number:	INT := 0;
	i:		INT;
	sum:	REAL;
END_VAR

fbCycle(IN:= NOT fbCycle.Q,
		PT:= PT);

// write the current value into the buffer		
buffer[index] := IN;

// increase the index
IF index < 30000 THEN
	index := index + 1;
END_IF

Overflow := (index = 30000);

// during the first cycle number will be smaller than index
IF number < index THEN
	number := index;
END_IF

// sum up the buffer to the current number
sum := 0.0;
MINAVG := IN;
MAXAVG := IN;
FOR i :=0 TO number-1 DO
	sum := sum + buffer[i];
	MINAVG := MIN(buffer[i], MINAVG);
	MAXAVG := MAX(buffer[i], MAXAVG);
END_FOR

// return the average
AVG := sum / number;

// if we hit the cycle time, reset the index and overwrite old values
IF fbCycle.Q THEN
	number := index;
	index := 0;
END_IF

END_FUNCTION_BLOCK

// ---- GlobalTextList.TcGTLO
TEXTLIST GlobalTextList
  272 = 'busy'
  879 = 'Error'
  548 = 'GoHome'
  867 = 'GoTo'
  273 = 'park'
  919 = 'Power'
  120 = 'ready'
  685 = 'Reset'
  777 = 'slew'
  717 = 'sliding'
  572 = 'Stop'
  155 = 'stopped'
  362 = 'track'
  364 = 'tracking'
END_TEXTLIST

// ---- VISUs/Visualization.TcVIS
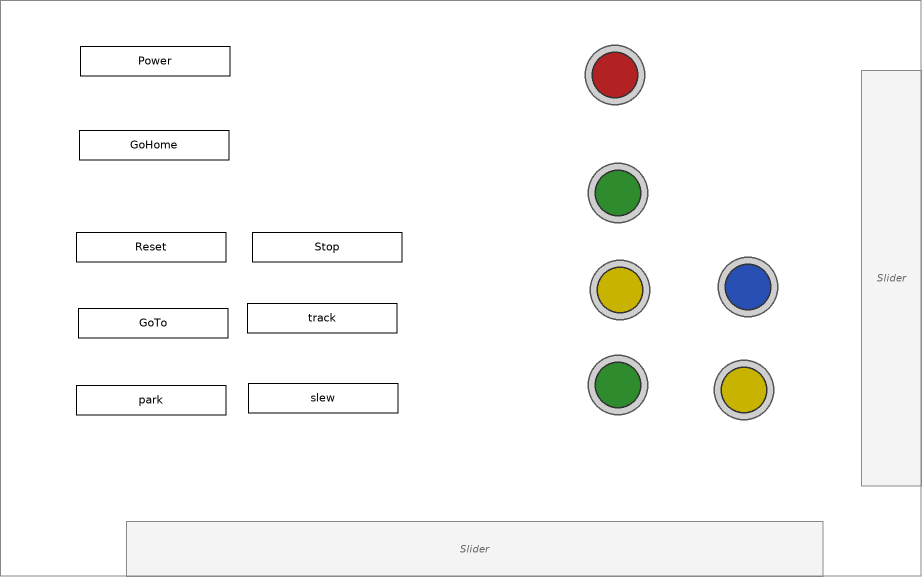
VISUALIZATION Visualization  // 922x577
    RoundedRectangle (80,46 150x30), "Power", colour toggle: TelescopeControl.power
        toggle TelescopeControl.power
    Rectangle (79,130 150x30), "GoHome", colour toggle: TelescopeControl.gohome
        toggle TelescopeControl.gohome
    Lamp1 (580,40 70x70), tooltip "Error", variable: TelescopeControl.error, style: Lamp-Lamp1-Red
    Lamp1 (583,158 70x70), tooltip "ready", variable: TelescopeControl.ready, style: Lamp-Lamp1-Green
    Rectangle (76,232 150x30), "Reset", colour toggle: TelescopeControl.reset
        toggle TelescopeControl.reset
    RoundedRectangle (78,308 150x30), "GoTo", colour toggle: TelescopeControl.goto
        toggle TelescopeControl.goto
    Lamp1 (585,255 70x70), tooltip "sliding", variable: TelescopeControl.sliding, style: Lamp-Lamp1-Yellow
    RoundedRectangle (76,385 150x30), "park", colour toggle: TelescopeControl.park
        toggle TelescopeControl.park
    Lamp1 (583,350 70x70), tooltip "stopped", variable: TelescopeControl.stopped, style: Lamp-Lamp1-Green
    Slider (126,521 697x56), variable: TelescopeControl.rightascension, scale 0..360
    Slider (861,70 61x416), variable: TelescopeControl.declination, scale -90..90
    Lamp1 (713,252 70x70), tooltip "tracking", variable: TelescopeControl.tracking, style: Lamp-Lamp1-Blue
    RoundedRectangle (247,303 150x30), "track", colour toggle: TelescopeControl.track
        toggle TelescopeControl.track
    RoundedRectangle (248,383 150x30), "slew", colour toggle: TelescopeControl.slew
        toggle TelescopeControl.slew
    Lamp1 (709,355 70x70), tooltip "busy", variable: TelescopeControl.busy, style: Lamp-Lamp1-Yellow
    RoundedRectangle (252,232 150x30), "Stop", colour toggle: TelescopeControl.stop
        toggle TelescopeControl.stop
END_VISUALIZATION
